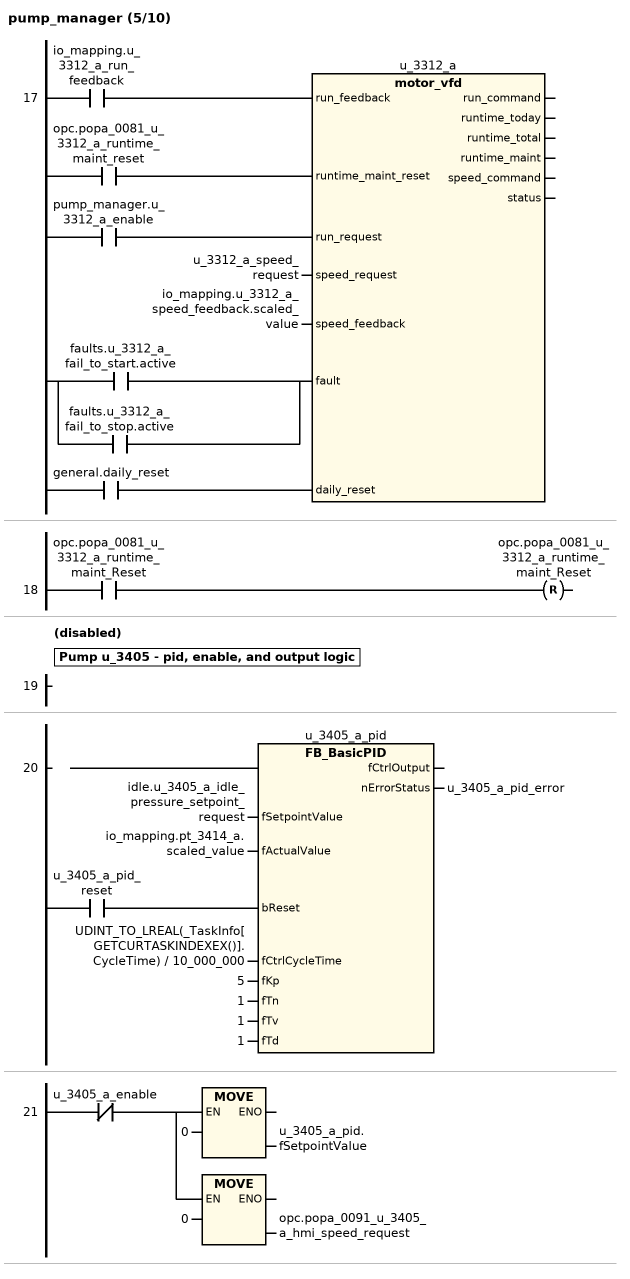
// NETWORK 17
u_3312_a(
    run_feedback := io_mapping.u_3312_a_run_feedback,
    runtime_maint_reset := opc.popa_0081_u_3312_a_runtime_maint_reset,
    run_request := pump_manager.u_3312_a_enable,
    speed_request := u_3312_a_speed_request,
    speed_feedback := io_mapping.u_3312_a_speed_feedback.scaled_value,
    fault := faults.u_3312_a_fail_to_start.active OR faults.u_3312_a_fail_to_stop.active,
    daily_reset := general.daily_reset); // motor_vfd

// NETWORK 18
opc.popa_0081_u_3312_a_runtime_maint_Reset R= opc.popa_0081_u_3312_a_runtime_maint_Reset;

// NETWORK 19 (disabled)
// label: Pump u_3405 - pid, enable, and output logic

// NETWORK 20
u_3405_a_pid(
    fSetpointValue := idle.u_3405_a_idle_pressure_setpoint_request,
    fActualValue := io_mapping.pt_3414_a.scaled_value,
    bReset := u_3405_a_pid_reset,
    fCtrlCycleTime := UDINT_TO_LREAL(_TaskInfo[GETCURTASKINDEXEX()].CycleTime) / 10_000_000,
    fKp := 5,
    fTn := 1,
    fTv := 1,
    fTd := 1,
    nErrorStatus => u_3405_a_pid_error); // FB_BasicPID

// NETWORK 21
_w16 := NOT u_3405_a_enable;
IF _w16 THEN u_3405_a_pid.fSetpointValue := 0; END_IF
IF _w16 THEN opc.popa_0091_u_3405_a_hmi_speed_request := 0; END_IF

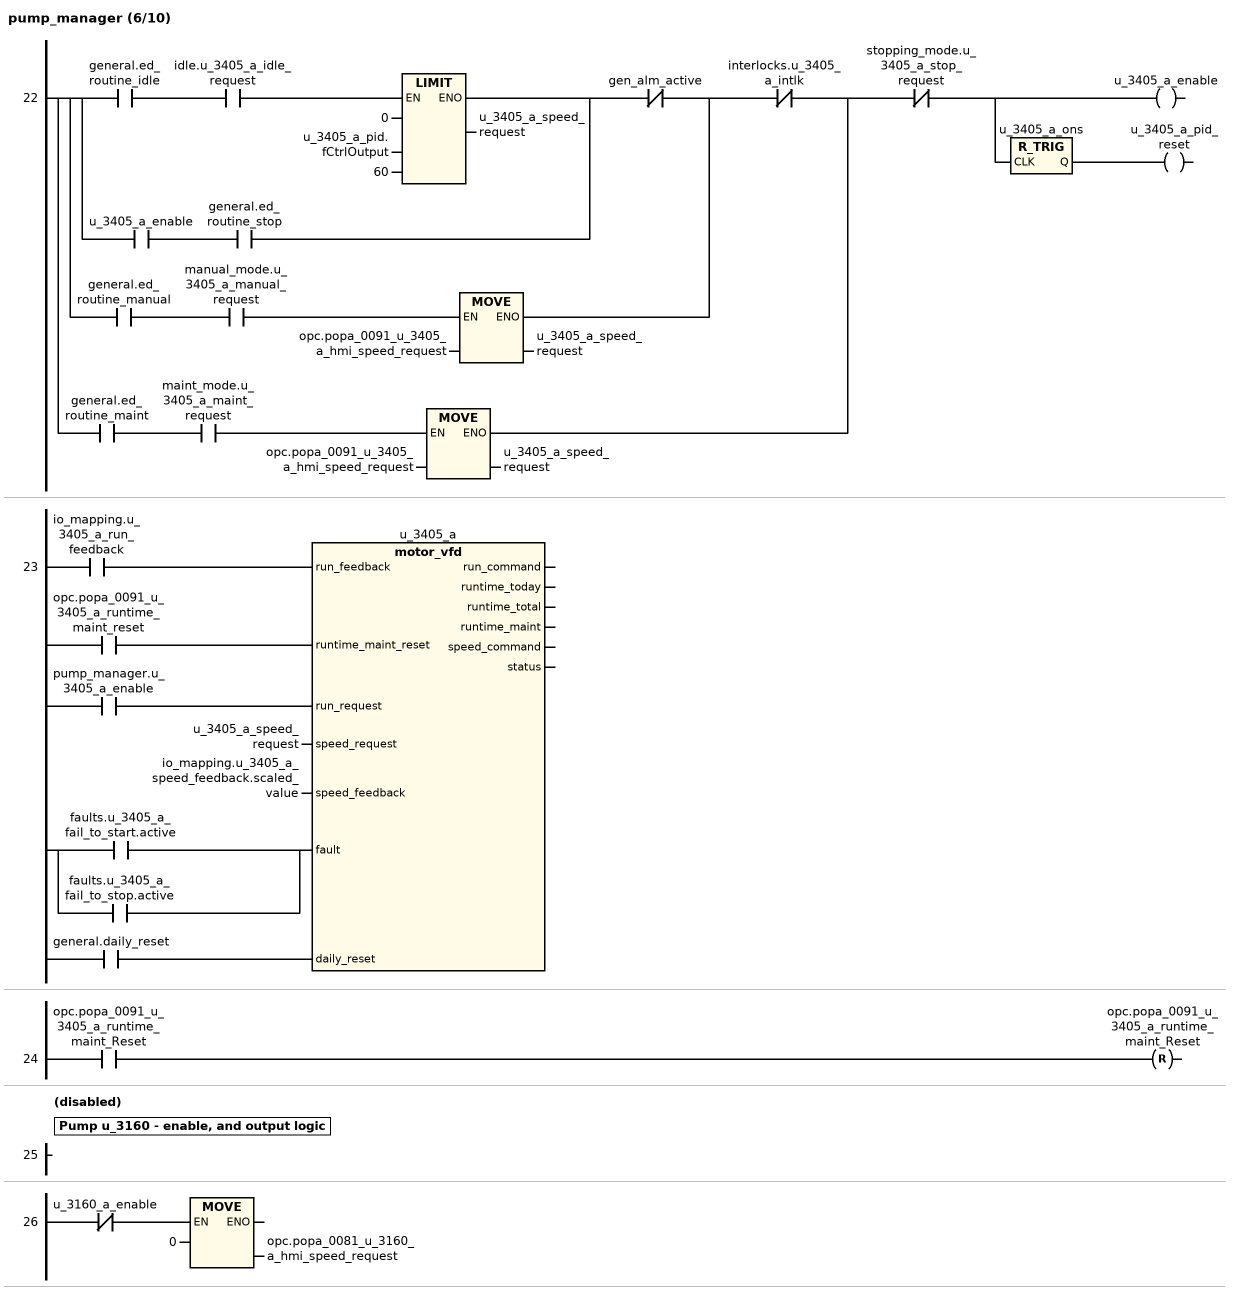
// NETWORK 22
_w17 := general.ed_routine_idle AND idle.u_3405_a_idle_request;
IF _w17 THEN u_3405_a_speed_request := LIMIT(0, u_3405_a_pid.fCtrlOutput, 60); END_IF
_w18 := general.ed_routine_manual AND manual_mode.u_3405_a_manual_request;
IF _w18 THEN u_3405_a_speed_request := opc.popa_0091_u_3405_a_hmi_speed_request; END_IF
_w19 := general.ed_routine_maint AND maint_mode.u_3405_a_maint_request;
IF _w19 THEN u_3405_a_speed_request := opc.popa_0091_u_3405_a_hmi_speed_request; END_IF
_w20 := (((_w17 OR u_3405_a_enable AND general.ed_routine_stop) AND NOT gen_alm_active OR _w18) AND NOT interlocks.u_3405_a_intlk OR _w19) AND NOT stopping_mode.u_3405_a_stop_request;
u_3405_a_enable := _w20;
u_3405_a_ons(CLK := _w20); // R_TRIG
u_3405_a_pid_reset := u_3405_a_ons.Q;

// NETWORK 23
u_3405_a(
    run_feedback := io_mapping.u_3405_a_run_feedback,
    runtime_maint_reset := opc.popa_0091_u_3405_a_runtime_maint_reset,
    run_request := pump_manager.u_3405_a_enable,
    speed_request := u_3405_a_speed_request,
    speed_feedback := io_mapping.u_3405_a_speed_feedback.scaled_value,
    fault := faults.u_3405_a_fail_to_start.active OR faults.u_3405_a_fail_to_stop.active,
    daily_reset := general.daily_reset); // motor_vfd

// NETWORK 24
opc.popa_0091_u_3405_a_runtime_maint_Reset R= opc.popa_0091_u_3405_a_runtime_maint_Reset;

// NETWORK 25 (disabled)
// label: Pump u_3160 - enable, and output logic

// NETWORK 26
IF NOT u_3160_a_enable THEN opc.popa_0081_u_3160_a_hmi_speed_request := 0; END_IF

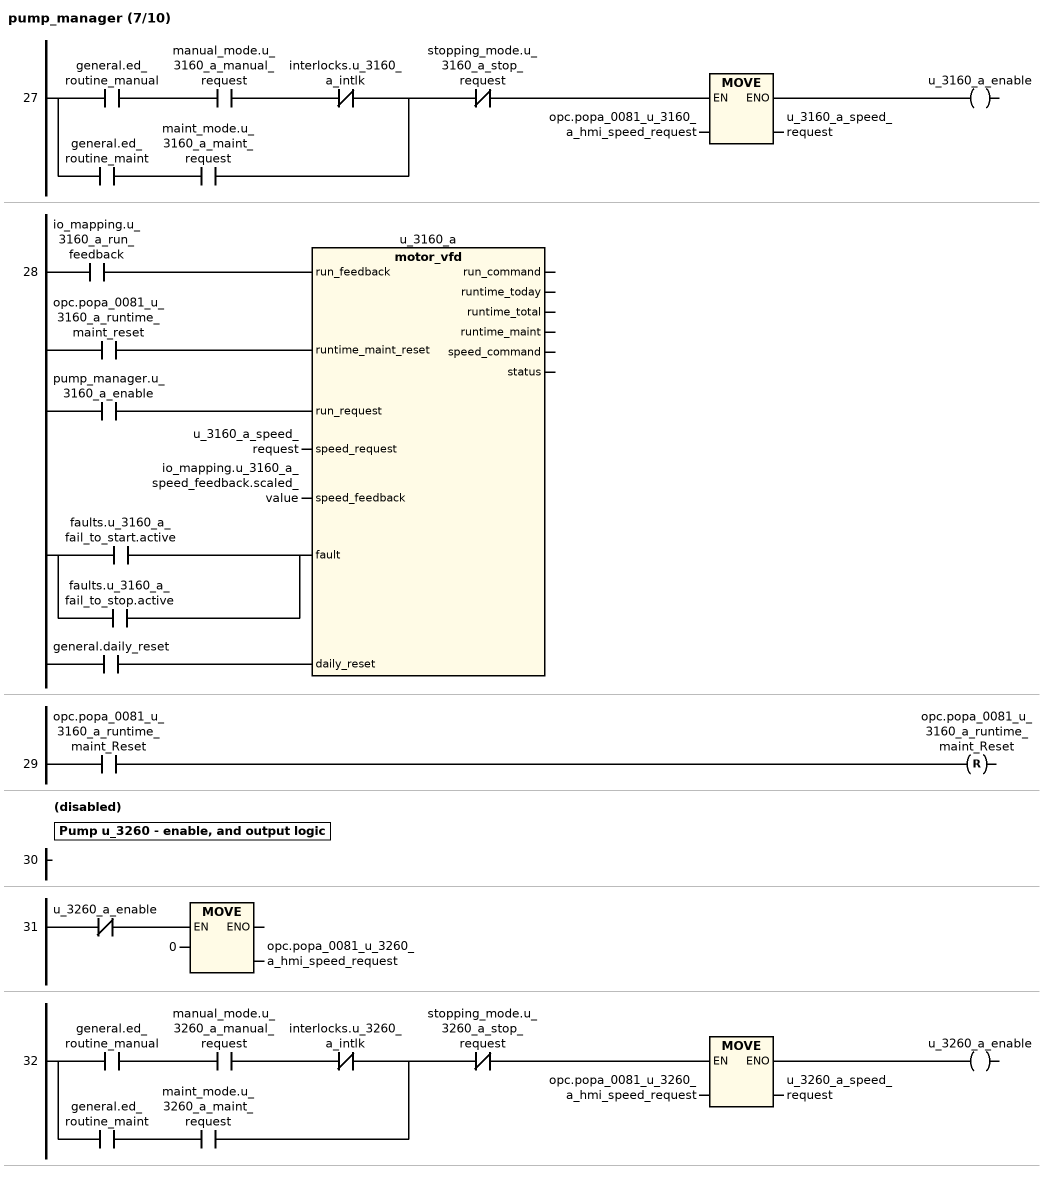
// NETWORK 27
_w21 := (general.ed_routine_manual AND manual_mode.u_3160_a_manual_request AND NOT interlocks.u_3160_a_intlk OR general.ed_routine_maint AND maint_mode.u_3160_a_maint_request) AND NOT stopping_mode.u_3160_a_stop_request;
IF _w21 THEN u_3160_a_speed_request := opc.popa_0081_u_3160_a_hmi_speed_request; END_IF
u_3160_a_enable := _w21;

// NETWORK 28
u_3160_a(
    run_feedback := io_mapping.u_3160_a_run_feedback,
    runtime_maint_reset := opc.popa_0081_u_3160_a_runtime_maint_reset,
    run_request := pump_manager.u_3160_a_enable,
    speed_request := u_3160_a_speed_request,
    speed_feedback := io_mapping.u_3160_a_speed_feedback.scaled_value,
    fault := faults.u_3160_a_fail_to_start.active OR faults.u_3160_a_fail_to_stop.active,
    daily_reset := general.daily_reset); // motor_vfd

// NETWORK 29
opc.popa_0081_u_3160_a_runtime_maint_Reset R= opc.popa_0081_u_3160_a_runtime_maint_Reset;

// NETWORK 30 (disabled)
// label: Pump u_3260 - enable, and output logic

// NETWORK 31
IF NOT u_3260_a_enable THEN opc.popa_0081_u_3260_a_hmi_speed_request := 0; END_IF

// NETWORK 32
_w22 := (general.ed_routine_manual AND manual_mode.u_3260_a_manual_request AND NOT interlocks.u_3260_a_intlk OR general.ed_routine_maint AND maint_mode.u_3260_a_maint_request) AND NOT stopping_mode.u_3260_a_stop_request;
IF _w22 THEN u_3260_a_speed_request := opc.popa_0081_u_3260_a_hmi_speed_request; END_IF
u_3260_a_enable := _w22;

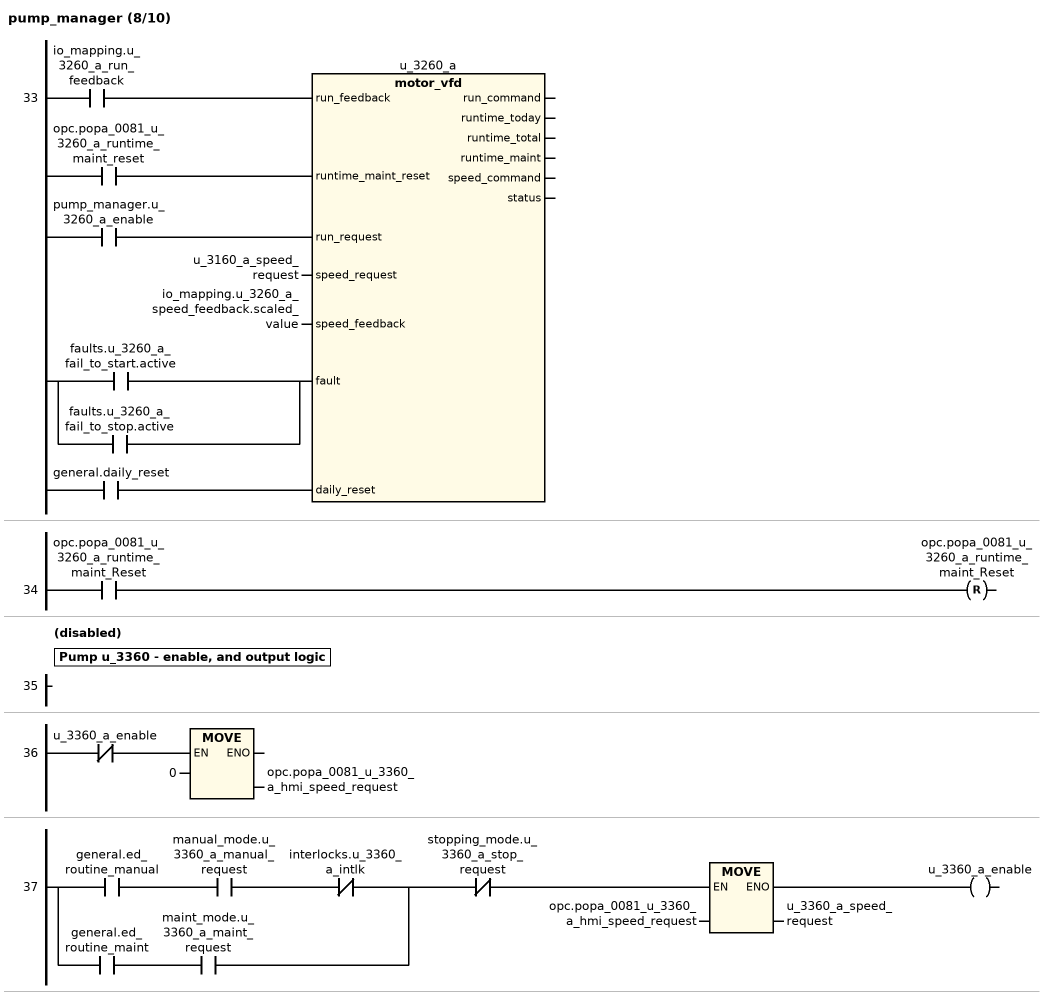
// NETWORK 33
u_3260_a(
    run_feedback := io_mapping.u_3260_a_run_feedback,
    runtime_maint_reset := opc.popa_0081_u_3260_a_runtime_maint_reset,
    run_request := pump_manager.u_3260_a_enable,
    speed_request := u_3160_a_speed_request,
    speed_feedback := io_mapping.u_3260_a_speed_feedback.scaled_value,
    fault := faults.u_3260_a_fail_to_start.active OR faults.u_3260_a_fail_to_stop.active,
    daily_reset := general.daily_reset); // motor_vfd

// NETWORK 34
opc.popa_0081_u_3260_a_runtime_maint_Reset R= opc.popa_0081_u_3260_a_runtime_maint_Reset;

// NETWORK 35 (disabled)
// label: Pump u_3360 - enable, and output logic

// NETWORK 36
IF NOT u_3360_a_enable THEN opc.popa_0081_u_3360_a_hmi_speed_request := 0; END_IF

// NETWORK 37
_w23 := (general.ed_routine_manual AND manual_mode.u_3360_a_manual_request AND NOT interlocks.u_3360_a_intlk OR general.ed_routine_maint AND maint_mode.u_3360_a_maint_request) AND NOT stopping_mode.u_3360_a_stop_request;
IF _w23 THEN u_3360_a_speed_request := opc.popa_0081_u_3360_a_hmi_speed_request; END_IF
u_3360_a_enable := _w23;

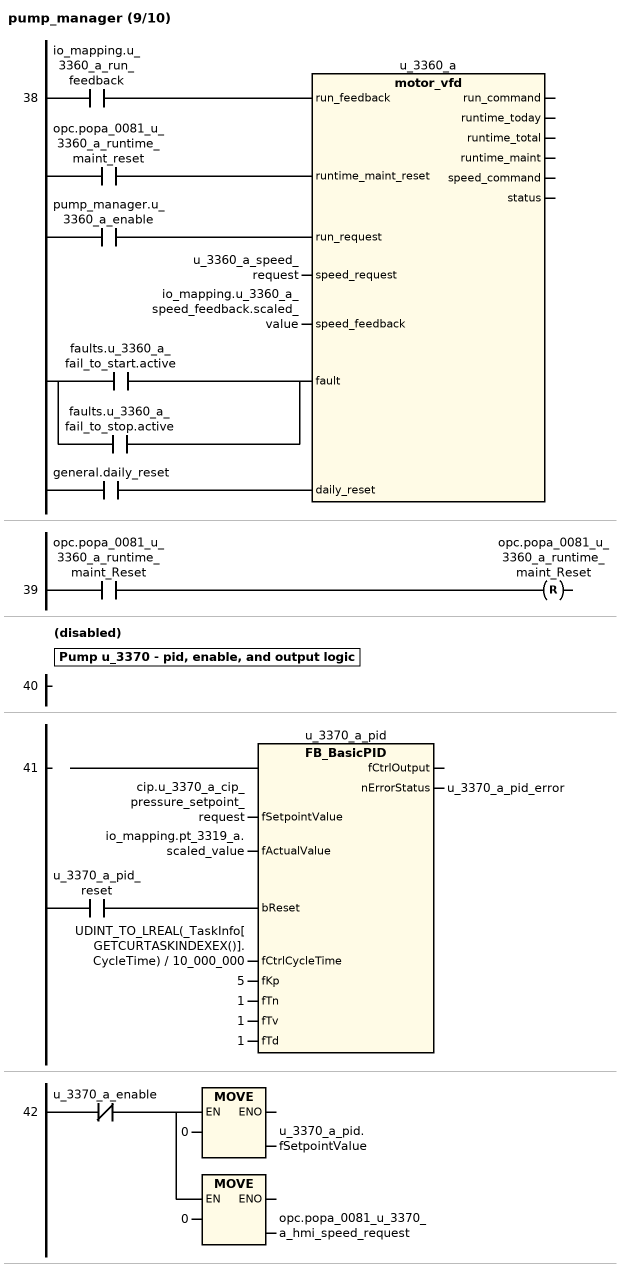
// NETWORK 38
u_3360_a(
    run_feedback := io_mapping.u_3360_a_run_feedback,
    runtime_maint_reset := opc.popa_0081_u_3360_a_runtime_maint_reset,
    run_request := pump_manager.u_3360_a_enable,
    speed_request := u_3360_a_speed_request,
    speed_feedback := io_mapping.u_3360_a_speed_feedback.scaled_value,
    fault := faults.u_3360_a_fail_to_start.active OR faults.u_3360_a_fail_to_stop.active,
    daily_reset := general.daily_reset); // motor_vfd

// NETWORK 39
opc.popa_0081_u_3360_a_runtime_maint_Reset R= opc.popa_0081_u_3360_a_runtime_maint_Reset;

// NETWORK 40 (disabled)
// label: Pump u_3370 - pid, enable, and output logic

// NETWORK 41
u_3370_a_pid(
    fSetpointValue := cip.u_3370_a_cip_pressure_setpoint_request,
    fActualValue := io_mapping.pt_3319_a.scaled_value,
    bReset := u_3370_a_pid_reset,
    fCtrlCycleTime := UDINT_TO_LREAL(_TaskInfo[GETCURTASKINDEXEX()].CycleTime) / 10_000_000,
    fKp := 5,
    fTn := 1,
    fTv := 1,
    fTd := 1,
    nErrorStatus => u_3370_a_pid_error); // FB_BasicPID

// NETWORK 42
_w24 := NOT u_3370_a_enable;
IF _w24 THEN u_3370_a_pid.fSetpointValue := 0; END_IF
IF _w24 THEN opc.popa_0081_u_3370_a_hmi_speed_request := 0; END_IF

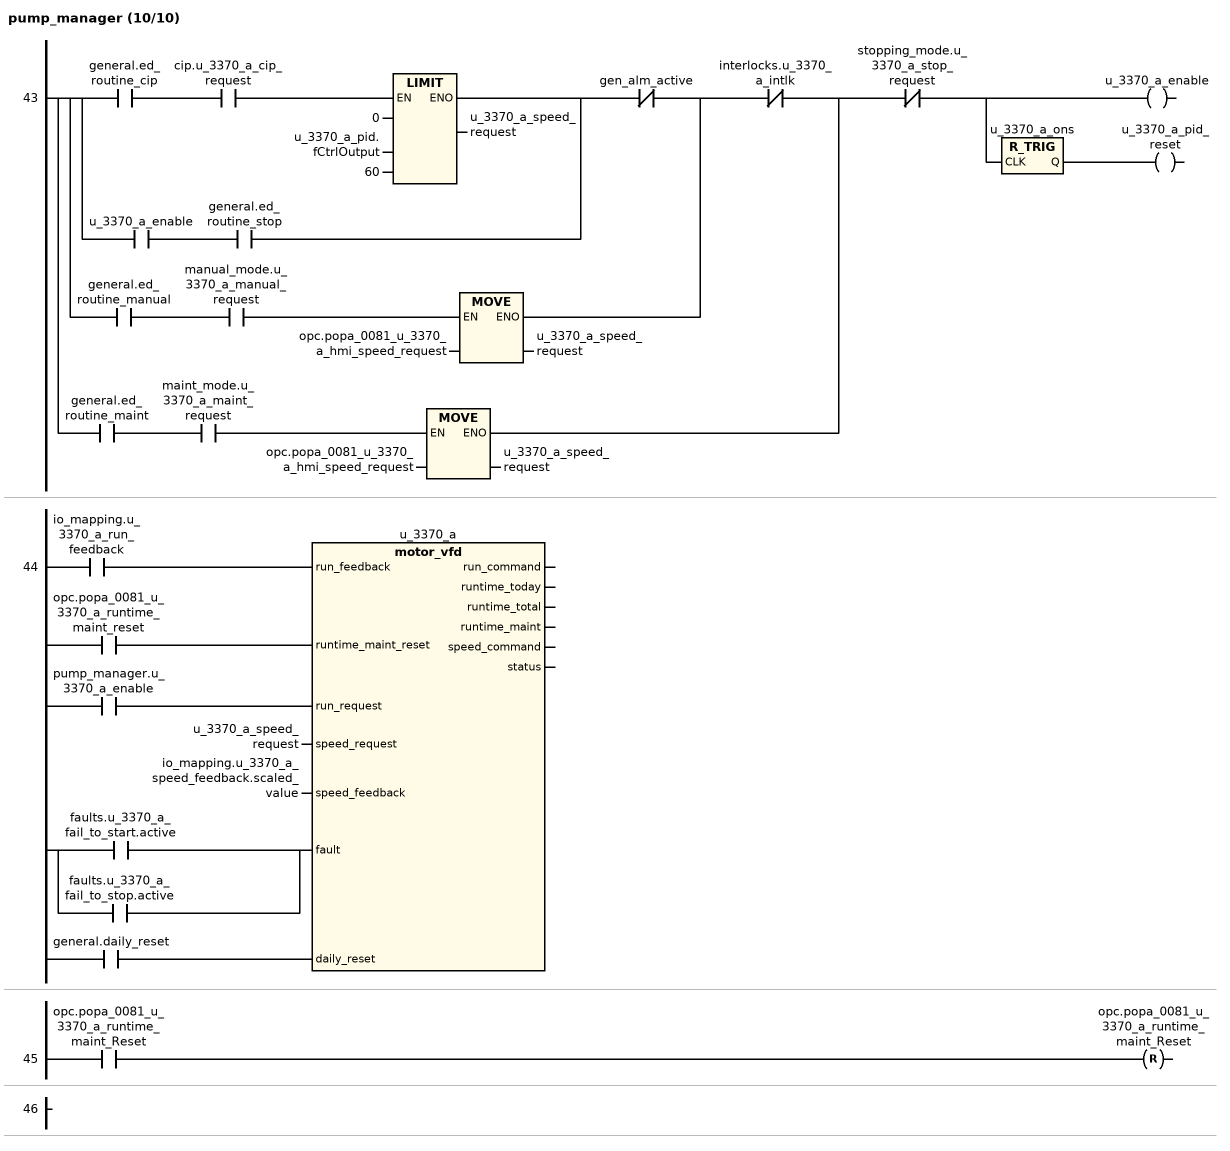
// NETWORK 43
_w25 := general.ed_routine_cip AND cip.u_3370_a_cip_request;
IF _w25 THEN u_3370_a_speed_request := LIMIT(0, u_3370_a_pid.fCtrlOutput, 60); END_IF
_w26 := general.ed_routine_manual AND manual_mode.u_3370_a_manual_request;
IF _w26 THEN u_3370_a_speed_request := opc.popa_0081_u_3370_a_hmi_speed_request; END_IF
_w27 := general.ed_routine_maint AND maint_mode.u_3370_a_maint_request;
IF _w27 THEN u_3370_a_speed_request := opc.popa_0081_u_3370_a_hmi_speed_request; END_IF
_w28 := (((_w25 OR u_3370_a_enable AND general.ed_routine_stop) AND NOT gen_alm_active OR _w26) AND NOT interlocks.u_3370_a_intlk OR _w27) AND NOT stopping_mode.u_3370_a_stop_request;
u_3370_a_enable := _w28;
u_3370_a_ons(CLK := _w28); // R_TRIG
u_3370_a_pid_reset := u_3370_a_ons.Q;

// NETWORK 44
u_3370_a(
    run_feedback := io_mapping.u_3370_a_run_feedback,
    runtime_maint_reset := opc.popa_0081_u_3370_a_runtime_maint_reset,
    run_request := pump_manager.u_3370_a_enable,
    speed_request := u_3370_a_speed_request,
    speed_feedback := io_mapping.u_3370_a_speed_feedback.scaled_value,
    fault := faults.u_3370_a_fail_to_start.active OR faults.u_3370_a_fail_to_stop.active,
    daily_reset := general.daily_reset); // motor_vfd

// NETWORK 45
opc.popa_0081_u_3370_a_runtime_maint_Reset R= opc.popa_0081_u_3370_a_runtime_maint_Reset;

// NETWORK 46

END_PROGRAM

// ---- POUs/idle.TcPOU
PROGRAM idle
VAR
	ed_routine_idle: BOOL;
	redox_doser_idle_enable: BOOL;
	
	tmr_idle_pumps: TON;
	u_3112_idle_request: BOOL;
	u_3312_idle_request: BOOL;
	u_3405_idle_request: BOOL;
	u_3212_idle_request: BOOL;
	tmr_idle_pump_delay: TON;
	u_3112_running: BOOL;
	u_3112_speed_ref: INT;
	u_3112_sp: REAL;
	salt_pressure_actual: REAL;
	u_3112_ready: BOOL;
	u_3212_running: BOOL;
	u_3212_ready: BOOL;
	u_3312_ready: BOOL;
	u_3312_running: BOOL;
	u_3405_running: BOOL;
	u_3405_ready: BOOL;
	stack_power_enable: BOOL;
	nv_3110_open_request: BOOL;
	nv_3210_open_request: BOOL;
	nv_3310_open_request: BOOL;
	nv_3110_open_feedback: BOOL;
	nv_3210_open_feedback: BOOL;
	nv_3310_open_feedback: BOOL;
	nv_3110_idle_request: BOOL;
	nv_3210_idle_request: BOOL;
	nv_3310_idle_request: BOOL;
	nv_3135_idle_request: BOOL;
	nv_3235_idle_request: BOOL;
	nv_3335_idle_request: BOOL;
	nv_3372_idle_request: BOOL;
	nv_3162_idle_request: BOOL;

	idle_stack_power_enable: BOOL;
	idle_TEMP_BIT: BOOL;
	tmr_idle_valye_delay: TON;
	tmr_idle_valve_delay: TON;
	tmr_idle_valve_delay_et: TIME;
	tmr_idle_valve_delay_pt: TIME := T#20S;
	tmr_idle_valve_delay_q: BOOL;
	u_3112_idle_pressure_setpoint_request: REAL;
	u_3212_idle_pressure_setpoint_request: REAL;
	u_3312_idle_pressure_setpoint_request: REAL;
	u_3405_idle_pressure_setpoint_request: REAL;
	idle_stable: BOOL;
	av_3148_idle_position_request: REAL;
	av_3248_idle_position_request: REAL;
	av_3348_idle_position_request: REAL;
	redox_pressure_calculation: REAL;
	redox_idle_pressure_sp_request: REAL;
	idle_startup_ons: R_TRIG;
END_VAR
VAR // added by the converter: edge detectors and wires of the graphical bodies
    _w1, _w2, _w3, _w4 : BOOL;
END_VAR

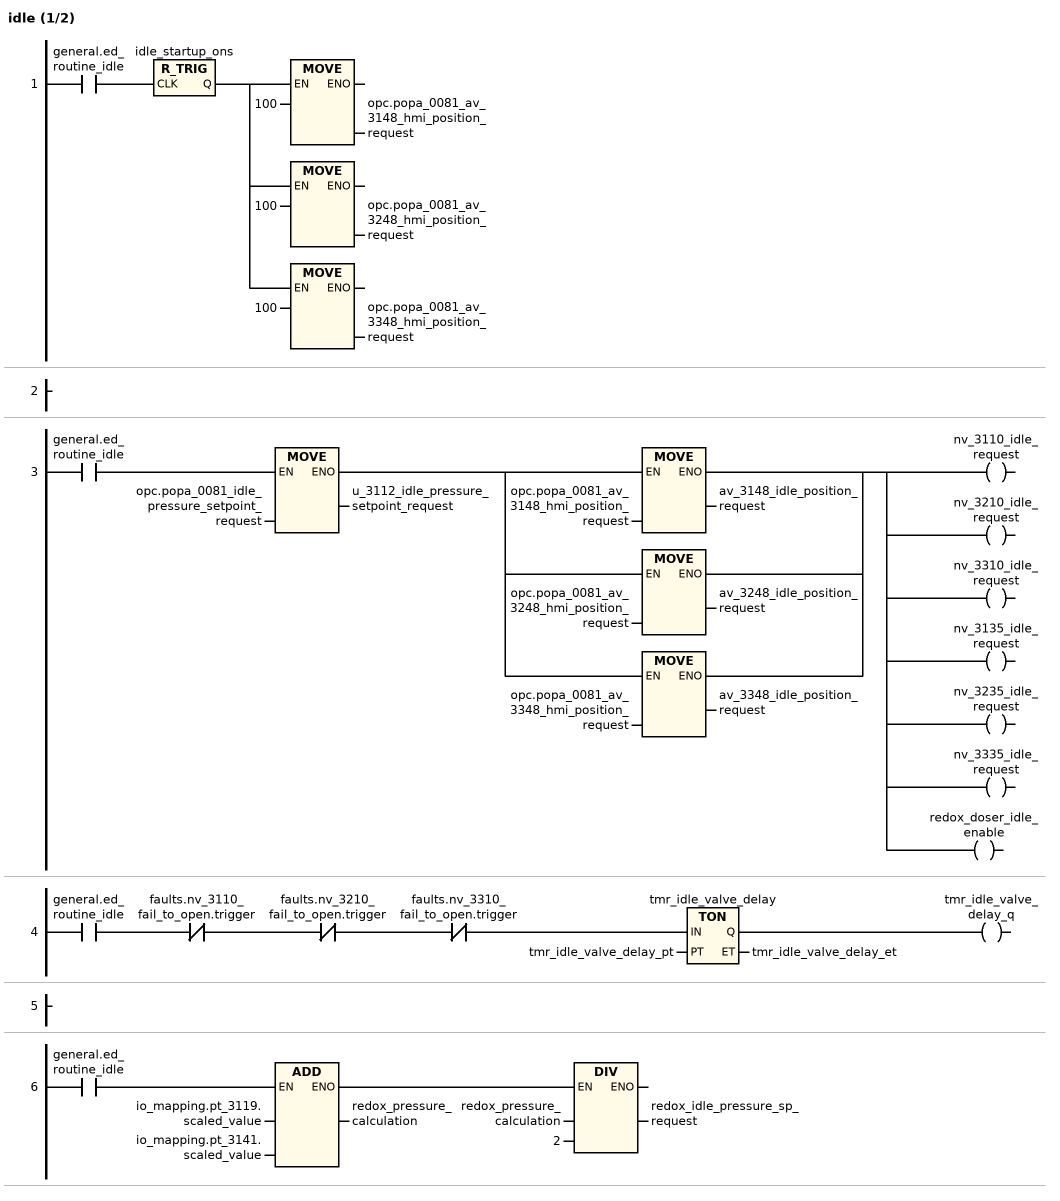
// NETWORK 1
idle_startup_ons(CLK := general.ed_routine_idle); // R_TRIG
IF idle_startup_ons.Q THEN opc.popa_0081_av_3148_hmi_position_request := 100; END_IF
IF idle_startup_ons.Q THEN opc.popa_0081_av_3248_hmi_position_request := 100; END_IF
IF idle_startup_ons.Q THEN opc.popa_0081_av_3348_hmi_position_request := 100; END_IF

// NETWORK 2

// NETWORK 3
_w1 := general.ed_routine_idle;
IF _w1 THEN u_3112_idle_pressure_setpoint_request := opc.popa_0081_idle_pressure_setpoint_request; END_IF
IF _w1 THEN av_3148_idle_position_request := opc.popa_0081_av_3148_hmi_position_request; END_IF
IF _w1 THEN av_3248_idle_position_request := opc.popa_0081_av_3248_hmi_position_request; END_IF
IF _w1 THEN av_3348_idle_position_request := opc.popa_0081_av_3348_hmi_position_request; END_IF
_w2 := _w1 OR (_w1 OR _w1);
nv_3110_idle_request := _w2;
nv_3210_idle_request := _w2;
nv_3310_idle_request := _w2;
nv_3135_idle_request := _w2;
nv_3235_idle_request := _w2;
nv_3335_idle_request := _w2;
redox_doser_idle_enable := _w2;

// NETWORK 4
tmr_idle_valve_delay(
    IN := general.ed_routine_idle AND NOT faults.nv_3110_fail_to_open.trigger AND NOT faults.nv_3210_fail_to_open.trigger AND NOT faults.nv_3310_fail_to_open.trigger,
    PT := tmr_idle_valve_delay_pt,
    ET => tmr_idle_valve_delay_et); // TON
tmr_idle_valve_delay_q := tmr_idle_valve_delay.Q;

// NETWORK 5

// NETWORK 6
_w3 := general.ed_routine_idle;
IF _w3 THEN redox_pressure_calculation := io_mapping.pt_3119.scaled_value + io_mapping.pt_3141.scaled_value; END_IF
IF _w3 THEN redox_idle_pressure_sp_request := redox_pressure_calculation / 2; END_IF

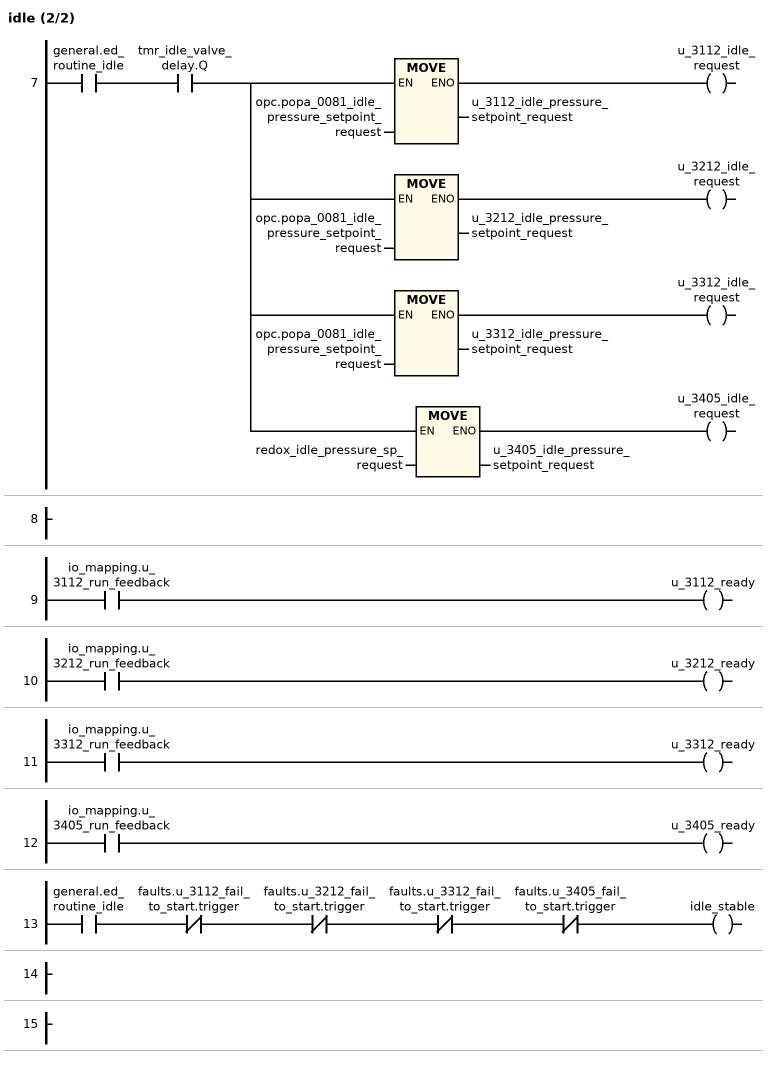
// NETWORK 7
_w4 := general.ed_routine_idle AND tmr_idle_valve_delay.Q;
IF _w4 THEN u_3112_idle_pressure_setpoint_request := opc.popa_0081_idle_pressure_setpoint_request; END_IF
u_3112_idle_request := _w4;
IF _w4 THEN u_3212_idle_pressure_setpoint_request := opc.popa_0081_idle_pressure_setpoint_request; END_IF
u_3212_idle_request := _w4;
IF _w4 THEN u_3312_idle_pressure_setpoint_request := opc.popa_0081_idle_pressure_setpoint_request; END_IF
u_3312_idle_request := _w4;
IF _w4 THEN u_3405_idle_pressure_setpoint_request := redox_idle_pressure_sp_request; END_IF
u_3405_idle_request := _w4;

// NETWORK 8

// NETWORK 9
u_3112_ready := io_mapping.u_3112_run_feedback;

// NETWORK 10
u_3212_ready := io_mapping.u_3212_run_feedback;

// NETWORK 11
u_3312_ready := io_mapping.u_3312_run_feedback;

// NETWORK 12
u_3405_ready := io_mapping.u_3405_run_feedback;

// NETWORK 13
idle_stable := general.ed_routine_idle AND NOT faults.u_3112_fail_to_start.trigger AND NOT faults.u_3212_fail_to_start.trigger AND NOT faults.u_3312_fail_to_start.trigger AND NOT faults.u_3405_fail_to_start.trigger;

// NETWORK 14

// NETWORK 15

END_PROGRAM

// ---- POUs/io_mapping.TcPOU
PROGRAM io_mapping
VAR PERSISTENT
//---Field Instrumentation-----------------------------------------------------------------------------------------------
    //Analog input function block
	cpt_3144_a: analog_scaling;
	
	cct_3120_a : analog_scaling;
	cct_3220_a : analog_scaling;
	cct_3320_a : analog_scaling;
	cct_3142_a : analog_scaling;
	cct_3242_a : analog_scaling;
	cct_3342_a : analog_scaling;
	
	ft_3122_a : analog_scaling;
	ft_3222_a : analog_scaling;
	ft_3322_a : analog_scaling;
	
	lt_3102_a : analog_scaling;
	lt_3202_a : analog_scaling;
	lt_3302_a : analog_scaling;
	lt_3153_a : analog_scaling;
	lt_3253_a : analog_scaling;
	lt_3353_a : analog_scaling;
	lt_3402_a : analog_scaling;
	
    pt_3119_a : analog_scaling;
	pt_3219_a : analog_scaling;
	pt_3319_a : analog_scaling;
	pt_3141_a : analog_scaling;
	pt_3241_a : analog_scaling;
	pt_3341_a : analog_scaling;
	pt_3428_a : analog_scaling;
	pt_3414_a : analog_scaling;
	
	tt_3118_a : analog_scaling;
	tt_3218_a : analog_scaling;
	tt_3318_a : analog_scaling;
	tt_3140_a : analog_scaling;
	tt_3240_a : analog_scaling;
	tt_3340_a : analog_scaling;
	tt_3432_a : analog_scaling;

	//Motor vfd speed feedback
	u_3112_a_speed_feedback : analog_scaling;
	u_3212_a_speed_feedback : analog_scaling;
	u_3312_a_speed_feedback : analog_scaling;
	u_3160_a_speed_feedback : analog_scaling;
	u_3260_a_speed_feedback : analog_scaling;
	u_3360_a_speed_feedback : analog_scaling;
	u_3370_a_speed_feedback : analog_scaling;
	u_3405_a_speed_feedback : analog_scaling;	
	
	//Analog valve position feedback
	av_3148_a_position_feedback : analog_scaling;
	av_3248_a_position_feedback : analog_scaling;
	av_3348_a_position_feedback : analog_scaling;
    //Analog input raw input, mapped to a physical input
    cpt_3144_a_raw_input AT %I* : INT;
	{attribute 'TcLinkTo' := 'TIID^Device 1 (EtherCAT)^Term 20 (EK1100-0018)^Term 24 (EL3058)^AI Standard Channel 1^Value'}
	cct_3120_a_raw_input AT %I* : INT;
	{attribute 'TcLinkTo' := 'TIID^Device 1 (EtherCAT)^Term 20 (EK1100-0018)^Term 24 (EL3058)^AI Standard Channel 2^Value'}
	cct_3220_a_raw_input AT %I* : INT;
	{attribute 'TcLinkTo' := 'TIID^Device 1 (EtherCAT)^Term 20 (EK1100-0018)^Term 24 (EL3058)^AI Standard Channel 3^Value'}
	cct_3320_a_raw_input AT %I* : INT;
	{attribute 'TcLinkTo' := 'TIID^Device 1 (EtherCAT)^Term 20 (EK1100-0018)^Term 24 (EL3058)^AI Standard Channel 4^Value'}
	cct_3142_a_raw_input AT %I* : INT;
	{attribute 'TcLinkTo' := 'TIID^Device 1 (EtherCAT)^Term 20 (EK1100-0018)^Term 24 (EL3058)^AI Standard Channel 5^Value'}
	cct_3242_a_raw_input AT %I* : INT;
	{attribute 'TcLinkTo' := 'TIID^Device 1 (EtherCAT)^Term 20 (EK1100-0018)^Term 24 (EL3058)^AI Standard Channel 6^Value'}
	cct_3342_a_raw_input AT %I* : INT;
	
	{attribute 'TcLinkTo' := 'TIID^Device 1 (EtherCAT)^Term 20 (EK1100-0018)^Term 25 (EL3058)^AI Standard Channel 1^Value'}
	ft_3122_a_raw_input AT %I* : INT;
	{attribute 'TcLinkTo' := 'TIID^Device 1 (EtherCAT)^Term 20 (EK1100-0018)^Term 25 (EL3058)^AI Standard Channel 2^Value'}
	ft_3222_a_raw_input AT %I* : INT;
	{attribute 'TcLinkTo' := 'TIID^Device 1 (EtherCAT)^Term 20 (EK1100-0018)^Term 25 (EL3058)^AI Standard Channel 3^Value'}
	ft_3322_a_raw_input AT %I* : INT;
	
	{attribute 'TcLinkTo' := 'TIID^Device 1 (EtherCAT)^Term 20 (EK1100-0018)^Term 21 (EL3058)^AI Standard Channel 1^Value'}
	pt_3119_a_raw_input AT %I* : INT;
	{attribute 'TcLinkTo' := 'TIID^Device 1 (EtherCAT)^Term 20 (EK1100-0018)^Term 21 (EL3058)^AI Standard Channel 2^Value'}
	pt_3219_a_raw_input AT %I* : INT;
	{attribute 'TcLinkTo' := 'TIID^Device 1 (EtherCAT)^Term 20 (EK1100-0018)^Term 21 (EL3058)^AI Standard Channel 3^Value'}
	pt_3319_a_raw_input AT %I* : INT;
	{attribute 'TcLinkTo' := 'TIID^Device 1 (EtherCAT)^Term 20 (EK1100-0018)^Term 21 (EL3058)^AI Standard Channel 4^Value'}
	pt_3141_a_raw_input AT %I* : INT;
	{attribute 'TcLinkTo' := 'TIID^Device 1 (EtherCAT)^Term 20 (EK1100-0018)^Term 21 (EL3058)^AI Standard Channel 5^Value'}
	pt_3241_a_raw_input AT %I* : INT;
	{attribute 'TcLinkTo' := 'TIID^Device 1 (EtherCAT)^Term 20 (EK1100-0018)^Term 21 (EL3058)^AI Standard Channel 6^Value'}
	pt_3341_a_raw_input AT %I* : INT;
	{attribute 'TcLinkTo' := 'TIID^Device 1 (EtherCAT)^Term 40 (EK1100)^Term 41 (EL3058)^AI Standard Channel 4^Value'}
	pt_3428_a_raw_input AT %I* : INT;
	{attribute 'TcLinkTo' := 'TIID^Device 1 (EtherCAT)^Term 40 (EK1100)^Term 41 (EL3058)^AI Standard Channel 5^Value'}
	pt_3414_a_raw_input AT %I* : INT;
	
	{attribute 'TcLinkTo' := 'TIID^Device 1 (EtherCAT)^Term 20 (EK1100-0018)^Term 23 (EL3058)^AI Standard Channel 3^Value'}
	lt_3102_a_raw_input AT %I* : INT;
	{attribute 'TcLinkTo' := 'TIID^Device 1 (EtherCAT)^Term 20 (EK1100-0018)^Term 23 (EL3058)^AI Standard Channel 4^Value'}
	lt_3202_a_raw_input AT %I* : INT;
	{attribute 'TcLinkTo' := 'TIID^Device 1 (EtherCAT)^Term 20 (EK1100-0018)^Term 23 (EL3058)^AI Standard Channel 5^Value'}
	lt_3302_a_raw_input AT %I* : INT;
	{attribute 'TcLinkTo' := 'TIID^Device 1 (EtherCAT)^Term 20 (EK1100-0018)^Term 23 (EL3058)^AI Standard Channel 6^Value'}
	lt_3153_a_raw_input AT %I* : INT;
	{attribute 'TcLinkTo' := 'TIID^Device 1 (EtherCAT)^Term 20 (EK1100-0018)^Term 23 (EL3058)^AI Standard Channel 7^Value'}
	lt_3253_a_raw_input AT %I* : INT;
	{attribute 'TcLinkTo' := 'TIID^Device 1 (EtherCAT)^Term 20 (EK1100-0018)^Term 23 (EL3058)^AI Standard Channel 8^Value'}
	lt_3353_a_raw_input AT %I* : INT;
	{attribute 'TcLinkTo' := 'TIID^Device 1 (EtherCAT)^Term 40 (EK1100)^Term 41 (EL3058)^AI Standard Channel 3^Value'}
	lt_3402_a_raw_input AT %I* : INT;
	
	{attribute 'TcLinkTo' := 'TIID^Device 1 (EtherCAT)^Term 20 (EK1100-0018)^Term 21 (EL3058)^AI Standard Channel 7^Value'}
	tt_3118_a_raw_input AT %I* : INT;
	{attribute 'TcLinkTo' := 'TIID^Device 1 (EtherCAT)^Term 20 (EK1100-0018)^Term 21 (EL3058)^AI Standard Channel 8^Value'}
	tt_3218_a_raw_input AT %I* : INT;
	{attribute 'TcLinkTo' := 'TIID^Device 1 (EtherCAT)^Term 20 (EK1100-0018)^Term 22 (EL3058)^AI Standard Channel 1^Value'}
	tt_3318_a_raw_input AT %I* : INT;
	{attribute 'TcLinkTo' := 'TIID^Device 1 (EtherCAT)^Term 20 (EK1100-0018)^Term 22 (EL3058)^AI Standard Channel 2^Value'}
	tt_3140_a_raw_input AT %I* : INT;
	{attribute 'TcLinkTo' := 'TIID^Device 1 (EtherCAT)^Term 20 (EK1100-0018)^Term 22 (EL3058)^AI Standard Channel 3^Value'}
	tt_3240_a_raw_input AT %I* : INT;
	{attribute 'TcLinkTo' := 'TIID^Device 1 (EtherCAT)^Term 20 (EK1100-0018)^Term 22 (EL3058)^AI Standard Channel 4^Value'}
	tt_3340_a_raw_input AT %I* : INT;
	{attribute 'TcLinkTo' := 'TIID^Device 1 (EtherCAT)^Term 40 (EK1100)^Term 41 (EL3058)^AI Standard Channel 2^Value'}
	tt_3432_a_raw_input AT %I* : INT;
	
//---Field Equipment:Pumps----------------------------------------------------------------------------------------------------------
	
	//Motor vfd run feedback, mapped to a physical input
	{attribute 'TcLinkTo' := 'TIID^Device 1 (EtherCAT)^Term 1 (EK1200)^Term 7 (EL1859)^Channel 2^Input'}
	u_3112_a_run_feedback AT %I* : BOOL;
	{attribute 'TcLinkTo' := 'TIID^Device 1 (EtherCAT)^Term 1 (EK1200)^Term 7 (EL1859)^Channel 4^Input'}
	u_3212_a_run_feedback AT %I* : BOOL;
	{attribute 'TcLinkTo' := 'TIID^Device 1 (EtherCAT)^Term 1 (EK1200)^Term 7 (EL1859)^Channel 6^Input'}
	u_3312_a_run_feedback AT %I* : BOOL;
	{attribute 'TcLinkTo' := 'TIID^Device 1 (EtherCAT)^Term 1 (EK1200)^Term 7 (EL1859)^Channel 8^Input'}
	u_3160_a_run_feedback AT %I* : BOOL;
	{attribute 'TcLinkTo' := 'TIID^Device 1 (EtherCAT)^Term 1 (EK1200)^Term 8 (EL1859)^Channel 2^Input'}
	u_3260_a_run_feedback AT %I* : BOOL;
	{attribute 'TcLinkTo' := 'TIID^Device 1 (EtherCAT)^Term 1 (EK1200)^Term 8 (EL1859)^Channel 4^Input'}
	u_3360_a_run_feedback AT %I* : BOOL;
	{attribute 'TcLinkTo' := 'TIID^Device 1 (EtherCAT)^Term 1 (EK1200)^Term 8 (EL1859)^Channel 6^Input'}
	u_3370_a_run_feedback AT %I* : BOOL;
	{attribute 'TcLinkTo' := 'TIID^Device 1 (EtherCAT)^Term 40 (EK1100)^Term 43 (EL1859)^Channel 2^Input'}
	u_3405_a_run_feedback AT %I* : BOOL;
	
	//Motor Fault feedback
	{attribute 'TcLinkTo' := 'TIID^Device 1 (EtherCAT)^Term 1 (EK1200)^Term 7 (EL1859)^Channel 1^Input'}
	u_3112_a_fault_feedback AT %I* : BOOL;
	{attribute 'TcLinkTo' := 'TIID^Device 1 (EtherCAT)^Term 1 (EK1200)^Term 7 (EL1859)^Channel 3^Input'}
	u_3212_a_fault_feedback AT %I* : BOOL;
	{attribute 'TcLinkTo' := 'TIID^Device 1 (EtherCAT)^Term 1 (EK1200)^Term 7 (EL1859)^Channel 5^Input'}
	u_3312_a_fault_feedback AT %I* : BOOL;
	{attribute 'TcLinkTo' := 'TIID^Device 1 (EtherCAT)^Term 1 (EK1200)^Term 7 (EL1859)^Channel 7^Input'}
	u_3160_a_fault_feedback AT %I* : BOOL;
	{attribute 'TcLinkTo' := 'TIID^Device 1 (EtherCAT)^Term 1 (EK1200)^Term 8 (EL1859)^Channel 1^Input'}
	u_3260_a_fault_feedback AT %I* : BOOL;
	{attribute 'TcLinkTo' := 'TIID^Device 1 (EtherCAT)^Term 1 (EK1200)^Term 8 (EL1859)^Channel 3^Input'}
	u_3360_a_fault_feedback AT %I* : BOOL;
	{attribute 'TcLinkTo' := 'TIID^Device 1 (EtherCAT)^Term 1 (EK1200)^Term 8 (EL1859)^Channel 5^Input'}
	u_3370_a_fault_feedback AT %I* : BOOL;
	{attribute 'TcLinkTo' := 'TIID^Device 1 (EtherCAT)^Term 40 (EK1100)^Term 43 (EL1859)^Channel 1^Input'}
	u_3405_a_fault_feedback AT %I* : BOOL;
	
	
	
	

	
	//Motor vfd speed feedback raw input
	{attribute 'TcLinkTo' := 'TIID^Device 1 (EtherCAT)^Term 1 (EK1200)^Term 2 (EL3058)^AI Standard Channel 1^Value'}
	u_3112_a_speed_feedback_raw_input AT %I* : INT;
	{attribute 'TcLinkTo' := 'TIID^Device 1 (EtherCAT)^Term 1 (EK1200)^Term 2 (EL3058)^AI Standard Channel 2^Value'}
	u_3212_a_speed_feedback_raw_input AT %I* : INT;
	{attribute 'TcLinkTo' := 'TIID^Device 1 (EtherCAT)^Term 1 (EK1200)^Term 2 (EL3058)^AI Standard Channel 3^Value'}
	u_3312_a_speed_feedback_raw_input AT %I* : INT;
	{attribute 'TcLinkTo' := 'TIID^Device 1 (EtherCAT)^Term 1 (EK1200)^Term 2 (EL3058)^AI Standard Channel 4^Value'}
	u_3160_a_speed_feedback_raw_input AT %I* : INT;
	{attribute 'TcLinkTo' := 'TIID^Device 1 (EtherCAT)^Term 1 (EK1200)^Term 2 (EL3058)^AI Standard Channel 5^Value'}
	u_3260_a_speed_feedback_raw_input AT %I* : INT;
	{attribute 'TcLinkTo' := 'TIID^Device 1 (EtherCAT)^Term 1 (EK1200)^Term 2 (EL3058)^AI Standard Channel 6^Value'}
	u_3360_a_speed_feedback_raw_input AT %I* : INT;
	{attribute 'TcLinkTo' := 'TIID^Device 1 (EtherCAT)^Term 1 (EK1200)^Term 2 (EL3058)^AI Standard Channel 7^Value'}
	u_3370_a_speed_feedback_raw_input AT %I* : INT;
	{attribute 'TcLinkTo' := 'TIID^Device 1 (EtherCAT)^Term 40 (EK1100)^Term 41 (EL3058)^AI Standard Channel 1^Value'}
	u_3405_a_speed_feedback_raw_input AT %I* : INT;
	
//--Field Equipent: Valves---------------------------------------------------------------------------------------------------------------
	

	//Analog valve position feedback raw input
	{attribute 'TcLinkTo' := 'TIID^Device 1 (EtherCAT)^Term 20 (EK1100-0018)^Term 22 (EL3058)^AI Standard Channel 8^Value'}
	av_3148_a_position_feedback_raw_input AT %I* : INT;
	{attribute 'TcLinkTo' := 'TIID^Device 1 (EtherCAT)^Term 20 (EK1100-0018)^Term 23 (EL3058)^AI Standard Channel 1^Value'}
	av_3248_a_position_feedback_raw_input AT %I* : INT;
	{attribute 'TcLinkTo' := 'TIID^Device 1 (EtherCAT)^Term 20 (EK1100-0018)^Term 23 (EL3058)^AI Standard Channel 2^Value'}
	av_3348_a_position_feedback_raw_input AT %I* : INT;
	

	
	//Digital valve open feedback
	//{attribute 'TcLinkTo' := 'TIID^Device 1 (EtherCAT)^Term 31 (EK1914)^Term 32 (EL1859)^Channel 11^Output'}
	nv_3110_a_open_feedback AT %I* : BOOL;
	//{attribute 'TcLinkTo' := 'TIID^Device 1 (EtherCAT)^Term 31 (EK1914)^Term 32 (EL1859)^Channel 11^Output'}
	nv_3210_a_open_feedback AT %I* : BOOL;
	//{attribute 'TcLinkTo' := 'TIID^Device 1 (EtherCAT)^Term 31 (EK1914)^Term 32 (EL1859)^Channel 11^Output'}
	nv_3310_a_open_feedback AT %I* : BOOL;
	{attribute 'TcLinkTo' := 'TIID^Device 1 (EtherCAT)^Term 20 (EK1100-0018)^Term 28 (EL1859)^Channel 1^Input'}
	nv_3135_a_open_feedback AT %I* : BOOL;
	{attribute 'TcLinkTo' := 'TIID^Device 1 (EtherCAT)^Term 20 (EK1100-0018)^Term 28 (EL1859)^Channel 2^Input'}
	nv_3235_a_open_feedback AT %I* : BOOL;
	{attribute 'TcLinkTo' := 'TIID^Device 1 (EtherCAT)^Term 20 (EK1100-0018)^Term 28 (EL1859)^Channel 3^Input'}
	nv_3335_a_open_feedback AT %I* : BOOL;
	{attribute 'TcLinkTo' := 'TIID^Device 1 (EtherCAT)^Term 20 (EK1100-0018)^Term 28 (EL1859)^Channel 4^Input'}
	nv_3372_a_open_feedback AT %I* : BOOL;
	{attribute 'TcLinkTo' := 'TIID^Device 1 (EtherCAT)^Term 20 (EK1100-0018)^Term 28 (EL1859)^Channel 5^Input'}
	nv_3162_a_open_feedback AT %I* : BOOL;
	
	//Digital valve closed feedback
	//{attribute 'TcLinkTo' := 'TIID^Device 1 (EtherCAT)^Term 31 (EK1914)^Term 32 (EL1859)^Channel 11^Output'}
	nv_3110_a_closed_feedback AT %I* : BOOL;
	//{attribute 'TcLinkTo' := 'TIID^Device 1 (EtherCAT)^Term 31 (EK1914)^Term 32 (EL1859)^Channel 11^Output'}
	nv_3210_a_closed_feedback AT %I* : BOOL;
	//{attribute 'TcLinkTo' := 'TIID^Device 1 (EtherCAT)^Term 31 (EK1914)^Term 32 (EL1859)^Channel 11^Output'}
	nv_3310_a_closed_feedback AT %I* : BOOL;
	{attribute 'TcLinkTo' := 'TIID^Device 1 (EtherCAT)^Term 20 (EK1100-0018)^Term 29 (EL1859)^Channel 1^Input'}
	nv_3135_a_closed_feedback AT %I* : BOOL;
	{attribute 'TcLinkTo' := 'TIID^Device 1 (EtherCAT)^Term 20 (EK1100-0018)^Term 29 (EL1859)^Channel 2^Input'}
	nv_3235_a_closed_feedback AT %I* : BOOL;
	{attribute 'TcLinkTo' := 'TIID^Device 1 (EtherCAT)^Term 20 (EK1100-0018)^Term 29 (EL1859)^Channel 3^Input'}
	nv_3335_a_closed_feedback AT %I* : BOOL;
	{attribute 'TcLinkTo' := 'TIID^Device 1 (EtherCAT)^Term 20 (EK1100-0018)^Term 29 (EL1859)^Channel 4^Input'}
	nv_3372_a_closed_feedback AT %I* : BOOL;
	{attribute 'TcLinkTo' := 'TIID^Device 1 (EtherCAT)^Term 20 (EK1100-0018)^Term 29 (EL1859)^Channel 5^Input'}
	nv_3162_a_closed_feedback AT %I* : BOOL;
	

END_VAR

//---Field Instrumentation--------------------------------------------------------------------------------------------------

//Instantiate analog input function block
cpt_3144_a();
//Map values from the OPC GVL so that they can be written to from outside POU(IE from HMI)
cpt_3144_a.eu_max:=opc.popa_0081_cpt_3144_a_eu_max;
cpt_3144_a.eu_min:=opc.popa_0081_cpt_3144_a_eu_min;
cpt_3144_a.filter_factor:=opc.popa_0081_cpt_3144_a_filter_factor;
cpt_3144_a.raw_max:=opc.popa_0081_cpt_3144_a_raw_max;
cpt_3144_a.raw_min:=opc.popa_0081_cpt_3144_a_raw_min;
//Map the analog scaling function block raw input to the physical raw input variable
cpt_3144_a.raw_input := cpt_3144_a_raw_input;

//Instantiate analog input function block
cct_3120_a();
//Map values from the OPC GVL so that they can be written to from outside POU(IE from HMI)
cct_3120_a.eu_max:=opc.popa_0081_cct_3120_a_eu_max;
cct_3120_a.eu_min:=opc.popa_0081_cct_3120_a_eu_min;
cct_3120_a.filter_factor:=opc.popa_0081_cct_3120_a_filter_factor;
cct_3120_a.raw_max:=opc.popa_0081_cct_3120_a_raw_max;
cct_3120_a.raw_min:=opc.popa_0081_cct_3120_a_raw_min;
//Map the analog scaling function block raw input to the physical raw input variable
cct_3120_a.raw_input := cct_3120_a_raw_input;

//Instantiate analog input function block
cct_3220_a();
//Map values from the OPC GVL so that they can be written to from outside POU(IE from HMI)
cct_3220_a.eu_max:=opc.popa_0081_cct_3220_a_eu_max;
cct_3220_a.eu_min:=opc.popa_0081_cct_3220_a_eu_min;
cct_3220_a.filter_factor:=opc.popa_0081_cct_3220_a_filter_factor;
cct_3220_a.raw_max:=opc.popa_0081_cct_3220_a_raw_max;
cct_3220_a.raw_min:=opc.popa_0081_cct_3220_a_raw_min;
//Map the analog scaling function block raw input to the physical raw input variable
cct_3220_a.raw_input := cct_3220_a_raw_input;

//Instantiate analog input function block
cct_3320_a();
//Map values from the OPC GVL so that they can be written to from outside POU(IE from HMI)
cct_3320_a.eu_max:=opc.popa_0081_cct_3320_a_eu_max;
cct_3320_a.eu_min:=opc.popa_0081_cct_3320_a_eu_min;
cct_3320_a.filter_factor:=opc.popa_0081_cct_3320_a_filter_factor;
cct_3320_a.raw_max:=opc.popa_0081_cct_3320_a_raw_max;
cct_3320_a.raw_min:=opc.popa_0081_cct_3320_a_raw_min;
//Map the analog scaling function block raw input to the physical raw input variable
cct_3320_a.raw_input := cct_3320_a_raw_input;

//Instantiate analog input function block
cct_3142_a();
//Map values from the OPC GVL so that they can be written to from outside POU(IE from HMI)
cct_3142_a.eu_max:=opc.popa_0081_cct_3142_a_eu_max;
cct_3142_a.eu_min:=opc.popa_0081_cct_3142_a_eu_min;
cct_3142_a.filter_factor:=opc.popa_0081_cct_3142_a_filter_factor;
cct_3142_a.raw_max:=opc.popa_0081_cct_3142_a_raw_max;
cct_3142_a.raw_min:=opc.popa_0081_cct_3142_a_raw_min;
//Map the analog scaling function block raw input to the physical raw input variable
cct_3142_a.raw_input := cct_3142_a_raw_input;

//Instantiate analog input function block
cct_3242_a();
//Map values from the OPC GVL so that they can be written to from outside POU(IE from HMI)
cct_3242_a.eu_max:=opc.popa_0081_cct_3242_a_eu_max;
cct_3242_a.eu_min:=opc.popa_0081_cct_3242_a_eu_min;
cct_3242_a.filter_factor:=opc.popa_0081_cct_3242_a_filter_factor;
cct_3242_a.raw_max:=opc.popa_0081_cct_3242_a_raw_max;
cct_3242_a.raw_min:=opc.popa_0081_cct_3242_a_raw_min;
//Map the analog scaling function block raw input to the physical raw input variable
cct_3242_a.raw_input := cct_3242_a_raw_input;

//Instantiate analog input function block
cct_3342_a();
//Map values from the OPC GVL so that they can be written to from outside POU(IE from HMI)
cct_3342_a.eu_max:=opc.popa_0081_cct_3342_a_eu_max;
cct_3342_a.eu_min:=opc.popa_0081_cct_3342_a_eu_min;
cct_3342_a.filter_factor:=opc.popa_0081_cct_3342_a_filter_factor;
cct_3342_a.raw_max:=opc.popa_0081_cct_3342_a_raw_max;
cct_3342_a.raw_min:=opc.popa_0081_cct_3342_a_raw_min;
//Map the analog scaling function block raw input to the physical raw input variable
cct_3342_a.raw_input := cct_3342_a_raw_input;

//Instantiate analog input function block
ft_3122_a();
//Map values from the OPC GVL so that they can be written to from outside POU(IE from HMI)
ft_3122_a.eu_max:=500;//opc.popa_0081_ft_3122_a_eu_max;
ft_3122_a.eu_min:=opc.popa_0081_ft_3122_a_eu_min;
ft_3122_a.filter_factor:=opc.popa_0081_ft_3122_a_filter_factor;
ft_3122_a.raw_max:=opc.popa_0081_ft_3122_a_raw_max;
ft_3122_a.raw_min:=opc.popa_0081_ft_3122_a_raw_min;
//Map the analog scaling function block raw input to the physical raw input variable
ft_3122_a.raw_input := ft_3122_a_raw_input;

//Instantiate analog input function block
ft_3222_a();
//Map values from the OPC GVL so that they can be written to from outside POU(IE from HMI)
ft_3222_a.eu_max:=500;//opc.popa_0081_ft_3222_a_eu_max;
ft_3222_a.eu_min:=opc.popa_0081_ft_3222_a_eu_min;
ft_3222_a.filter_factor:=opc.popa_0081_ft_3222_a_filter_factor;
ft_3222_a.raw_max:=opc.popa_0081_ft_3222_a_raw_max;
ft_3222_a.raw_min:=opc.popa_0081_ft_3222_a_raw_min;
//Map the analog scaling function block raw input to the physical raw input variable
ft_3222_a.raw_input := ft_3222_a_raw_input;

//Instantiate analog input function block
ft_3322_a();
//Map values from the OPC GVL so that they can be written to from outside POU(IE from HMI)
ft_3322_a.eu_max:=500;//opc.popa_0081_ft_3322_a_eu_max;
ft_3322_a.eu_min:=opc.popa_0081_ft_3322_a_eu_min;
ft_3322_a.filter_factor:=opc.popa_0081_ft_3322_a_filter_factor;
ft_3322_a.raw_max:=opc.popa_0081_ft_3322_a_raw_max;
ft_3322_a.raw_min:=opc.popa_0081_ft_3322_a_raw_min;
//Map the analog scaling function block raw input to the physical raw input variable
ft_3322_a.raw_input := ft_3322_a_raw_input;

//Instantiate analog input function block
lt_3102_a();
//Map values from the OPC GVL so that they can be written to from outside POU(IE from HMI)
lt_3102_a.eu_max:=opc.popa_0081_lt_3102_a_eu_max;
lt_3102_a.eu_min:=opc.popa_0081_lt_3102_a_eu_min;
lt_3102_a.filter_factor:=opc.popa_0081_lt_3102_a_filter_factor;
lt_3102_a.raw_max:=opc.popa_0081_lt_3102_a_raw_max;
lt_3102_a.raw_min:=opc.popa_0081_lt_3102_a_raw_min;
//Map the analog scaling function block raw input to the physical raw input variable
lt_3102_a.raw_input := lt_3102_a_raw_input;

//Instantiate analog input function block
lt_3202_a();
//Map values from the OPC GVL so that they can be written to from outside POU(IE from HMI)
lt_3202_a.eu_max:=opc.popa_0081_lt_3202_a_eu_max;
lt_3202_a.eu_min:=opc.popa_0081_lt_3202_a_eu_min;
lt_3202_a.filter_factor:=opc.popa_0081_lt_3202_a_filter_factor;
lt_3202_a.raw_max:=opc.popa_0081_lt_3202_a_raw_max;
lt_3202_a.raw_min:=opc.popa_0081_lt_3202_a_raw_min;
//Map the analog scaling function block raw input to the physical raw input variable
lt_3202_a.raw_input := lt_3202_a_raw_input;

//Instantiate analog input function block
lt_3302_a();
//Map values from the OPC GVL so that they can be written to from outside POU(IE from HMI)
lt_3302_a.eu_max:=opc.popa_0081_lt_3302_a_eu_max;
lt_3302_a.eu_min:=opc.popa_0081_lt_3302_a_eu_min;
lt_3302_a.filter_factor:=opc.popa_0081_lt_3302_a_filter_factor;
lt_3302_a.raw_max:=opc.popa_0081_lt_3302_a_raw_max;
lt_3302_a.raw_min:=opc.popa_0081_lt_3302_a_raw_min;
//Map the analog scaling function block raw input to the physical raw input variable
lt_3302_a.raw_input := lt_3302_a_raw_input;

//Instantiate analog input function block
lt_3153_a();
//Map values from the OPC GVL so that they can be written to from outside POU(IE from HMI)
lt_3153_a.eu_max:=opc.popa_0081_lt_3153_a_eu_max;
lt_3153_a.eu_min:=opc.popa_0081_lt_3153_a_eu_min;
lt_3153_a.filter_factor:=opc.popa_0081_lt_3153_a_filter_factor;
lt_3153_a.raw_max:=opc.popa_0081_lt_3153_a_raw_max;
lt_3153_a.raw_min:=opc.popa_0081_lt_3153_a_raw_min;
//Map the analog scaling function block raw input to the physical raw input variable
lt_3153_a.raw_input := lt_3153_a_raw_input;

//Instantiate analog input function block
lt_3253_a();
//Map values from the OPC GVL so that they can be written to from outside POU(IE from HMI)
lt_3253_a.eu_max:=opc.popa_0081_lt_3253_a_eu_max;
lt_3253_a.eu_min:=opc.popa_0081_lt_3253_a_eu_min;
lt_3253_a.filter_factor:=opc.popa_0081_lt_3253_a_filter_factor;
lt_3253_a.raw_max:=opc.popa_0081_lt_3253_a_raw_max;
lt_3253_a.raw_min:=opc.popa_0081_lt_3253_a_raw_min;
//Map the analog scaling function block raw input to the physical raw input variable
lt_3253_a.raw_input := lt_3253_a_raw_input;

//Instantiate analog input function block
lt_3353_a();
//Map values from the OPC GVL so that they can be written to from outside POU(IE from HMI)
lt_3353_a.eu_max:=opc.popa_0081_lt_3353_a_eu_max;
lt_3353_a.eu_min:=opc.popa_0081_lt_3353_a_eu_min;
lt_3353_a.filter_factor:=opc.popa_0081_lt_3353_a_filter_factor;
lt_3353_a.raw_max:=opc.popa_0081_lt_3353_a_raw_max;
lt_3353_a.raw_min:=opc.popa_0081_lt_3353_a_raw_min;
//Map the analog scaling function block raw input to the physical raw input variable
lt_3353_a.raw_input := lt_3353_a_raw_input;

//Instantiate analog input function block
lt_3402_a();
//Map values from the OPC GVL so that they can be written to from outside POU(IE from HMI)
lt_3402_a.eu_max:=opc.popa_0091_lt_3402_a_eu_max;
lt_3402_a.eu_min:=opc.popa_0091_lt_3402_a_eu_min;
lt_3402_a.filter_factor:=opc.popa_0091_lt_3402_a_filter_factor;
lt_3402_a.raw_max:=opc.popa_0091_lt_3402_a_raw_max;
lt_3402_a.raw_min:=opc.popa_0091_lt_3402_a_raw_min;
//Map the analog scaling function block raw input to the physical raw input variable
lt_3402_a.raw_input := lt_3402_a_raw_input;

//Instantiate analog input function block
pt_3119_a();
//Map values from the OPC GVL so that they can be written to from outside POU(IE from HMI)
pt_3119_a.eu_max:=opc.popa_0081_pt_3119_a_eu_max;
pt_3119_a.eu_min:=opc.popa_0081_pt_3119_a_eu_min;
pt_3119_a.filter_factor:=opc.popa_0081_pt_3119_a_filter_factor;
pt_3119_a.raw_max:=opc.popa_0081_pt_3119_a_raw_max;
pt_3119_a.raw_min:=opc.popa_0081_pt_3119_a_raw_min;
//Map the analog scaling function block raw input to the physical raw input variable
pt_3119_a.raw_input := pt_3119_a_raw_input;

//Instantiate analog input function block
pt_3219_a();
//Map values from the OPC GVL so that they can be written to from outside POU(IE from HMI)
pt_3219_a.eu_max:=opc.popa_0081_pt_3219_a_eu_max;
pt_3219_a.eu_min:=opc.popa_0081_pt_3219_a_eu_min;
pt_3219_a.filter_factor:=opc.popa_0081_pt_3219_a_filter_factor;
pt_3219_a.raw_max:=opc.popa_0081_pt_3219_a_raw_max;
pt_3219_a.raw_min:=opc.popa_0081_pt_3219_a_raw_min;
//Map the analog scaling function block raw input to the physical raw input variable
pt_3219_a.raw_input := pt_3219_a_raw_input;

//Instantiate analog input function block
pt_3319_a();
//Map values from the OPC GVL so that they can be written to from outside POU(IE from HMI)
pt_3319_a.eu_max:=opc.popa_0081_pt_3319_a_eu_max;
pt_3319_a.eu_min:=opc.popa_0081_pt_3319_a_eu_min;
pt_3319_a.filter_factor:=opc.popa_0081_pt_3319_a_filter_factor;
pt_3319_a.raw_max:=opc.popa_0081_pt_3319_a_raw_max;
pt_3319_a.raw_min:=opc.popa_0081_pt_3319_a_raw_min;
//Map the analog scaling function block raw input to the physical raw input variable
pt_3319_a.raw_input := pt_3319_a_raw_input;

//Instantiate analog input function block
pt_3141_a();
//Map values from the OPC GVL so that they can be written to from outside POU(IE from HMI)
pt_3141_a.eu_max:=opc.popa_0081_pt_3141_a_eu_max;
pt_3141_a.eu_min:=opc.popa_0081_pt_3141_a_eu_min;
pt_3141_a.filter_factor:=opc.popa_0081_pt_3141_a_filter_factor;
pt_3141_a.raw_max:=opc.popa_0081_pt_3141_a_raw_max;
pt_3141_a.raw_min:=opc.popa_0081_pt_3141_a_raw_min;
//Map the analog scaling function block raw input to the physical raw input variable
pt_3141_a.raw_input := pt_3141_a_raw_input;

//Instantiate analog input function block
pt_3241_a();
//Map values from the OPC GVL so that they can be written to from outside POU(IE from HMI)
pt_3241_a.eu_max:=opc.popa_0081_pt_3241_a_eu_max;
pt_3241_a.eu_min:=opc.popa_0081_pt_3241_a_eu_min;
pt_3241_a.filter_factor:=opc.popa_0081_pt_3241_a_filter_factor;
pt_3241_a.raw_max:=opc.popa_0081_pt_3241_a_raw_max;
pt_3241_a.raw_min:=opc.popa_0081_pt_3241_a_raw_min;
//Map the analog scaling function block raw input to the physical raw input variable
pt_3241_a.raw_input := pt_3241_a_raw_input;

//Instantiate analog input function block
pt_3341_a();
//Map values from the OPC GVL so that they can be written to from outside POU(IE from HMI)
pt_3341_a.eu_max:=opc.popa_0081_pt_3341_a_eu_max;
pt_3341_a.eu_min:=opc.popa_0081_pt_3341_a_eu_min;
pt_3341_a.filter_factor:=opc.popa_0081_pt_3341_a_filter_factor;
pt_3341_a.raw_max:=opc.popa_0081_pt_3341_a_raw_max;
pt_3341_a.raw_min:=opc.popa_0081_pt_3341_a_raw_min;
//Map the analog scaling function block raw input to the physical raw input variable
pt_3341_a.raw_input := pt_3341_a_raw_input;

//Instantiate analog input function block
pt_3428_a();
//Map values from the OPC GVL so that they can be written to from outside POU(IE from HMI)
pt_3428_a.eu_max:=opc.popa_0091_pt_3428_a_eu_max;
pt_3428_a.eu_min:=opc.popa_0091_pt_3428_a_eu_min;
pt_3428_a.filter_factor:=opc.popa_0091_pt_3428_a_filter_factor;
pt_3428_a.raw_max:=opc.popa_0091_pt_3428_a_raw_max;
pt_3428_a.raw_min:=opc.popa_0091_pt_3428_a_raw_min;
//Map the analog scaling function block raw input to the physical raw input variable
pt_3428_a.raw_input := pt_3428_a_raw_input;

//Instantiate analog input function block
pt_3414_a();
//Map values from the OPC GVL so that they can be written to from outside POU(IE from HMI)
pt_3414_a.eu_max:=opc.popa_0091_pt_3414_a_eu_max;
pt_3414_a.eu_min:=opc.popa_0091_pt_3414_a_eu_min;
pt_3414_a.filter_factor:=opc.popa_0091_pt_3414_a_filter_factor;
pt_3414_a.raw_max:=opc.popa_0091_pt_3414_a_raw_max;
pt_3414_a.raw_min:=opc.popa_0091_pt_3414_a_raw_min;
//Map the analog scaling function block raw input to the physical raw input variable
pt_3414_a.raw_input := pt_3414_a_raw_input;

//Instantiate analog input function block
tt_3118_a();
//Map values from the OPC GVL so that they can be written to from outside POU(IE from HMI)
tt_3118_a.eu_max:=opc.popa_0081_tt_3118_a_eu_max;
tt_3118_a.eu_min:=opc.popa_0081_tt_3118_a_eu_min;
tt_3118_a.filter_factor:=opc.popa_0081_tt_3118_a_filter_factor;
tt_3118_a.raw_max:=opc.popa_0081_tt_3118_a_raw_max;
tt_3118_a.raw_min:=opc.popa_0081_tt_3118_a_raw_min;
//Map the analog scaling function block raw input to the physical raw input variable
tt_3118_a.raw_input := tt_3118_a_raw_input;

//Instantiate analog input function block
tt_3218_a();
//Map values from the OPC GVL so that they can be written to from outside POU(IE from HMI)
tt_3218_a.eu_max:=opc.popa_0081_tt_3218_a_eu_max;
tt_3218_a.eu_min:=opc.popa_0081_tt_3218_a_eu_min;
tt_3218_a.filter_factor:=opc.popa_0081_tt_3218_a_filter_factor;
tt_3218_a.raw_max:=opc.popa_0081_tt_3218_a_raw_max;
tt_3218_a.raw_min:=opc.popa_0081_tt_3218_a_raw_min;
//Map the analog scaling function block raw input to the physical raw input variable
tt_3218_a.raw_input := tt_3218_a_raw_input;

//Instantiate analog input function block
tt_3318_a();
//Map values from the OPC GVL so that they can be written to from outside POU(IE from HMI)
tt_3318_a.eu_max:=opc.popa_0081_tt_3318_a_eu_max;
tt_3318_a.eu_min:=opc.popa_0081_tt_3318_a_eu_min;
tt_3318_a.filter_factor:=opc.popa_0081_tt_3318_a_filter_factor;
tt_3318_a.raw_max:=opc.popa_0081_tt_3318_a_raw_max;
tt_3318_a.raw_min:=opc.popa_0081_tt_3318_a_raw_min;
//Map the analog scaling function block raw input to the physical raw input variable
tt_3318_a.raw_input := tt_3318_a_raw_input;

//Instantiate analog input function block
tt_3140_a();
//Map values from the OPC GVL so that they can be written to from outside POU(IE from HMI)
tt_3140_a.eu_max:=opc.popa_0081_tt_3140_a_eu_max;
tt_3140_a.eu_min:=opc.popa_0081_tt_3140_a_eu_min;
tt_3140_a.filter_factor:=opc.popa_0081_tt_3140_a_filter_factor;
tt_3140_a.raw_max:=opc.popa_0081_tt_3140_a_raw_max;
tt_3140_a.raw_min:=opc.popa_0081_tt_3140_a_raw_min;
//Map the analog scaling function block raw input to the physical raw input variable
tt_3140_a.raw_input := tt_3140_a_raw_input;

//Instantiate analog input function block
tt_3240_a();
//Map values from the OPC GVL so that they can be written to from outside POU(IE from HMI)
tt_3240_a.eu_max:=opc.popa_0081_tt_3240_a_eu_max;
tt_3240_a.eu_min:=opc.popa_0081_tt_3240_a_eu_min;
tt_3240_a.filter_factor:=opc.popa_0081_tt_3240_a_filter_factor;
tt_3240_a.raw_max:=opc.popa_0081_tt_3240_a_raw_max;
tt_3240_a.raw_min:=opc.popa_0081_tt_3240_a_raw_min;
//Map the analog scaling function block raw input to the physical raw input variable
tt_3240_a.raw_input := tt_3240_a_raw_input;

//Instantiate analog input function block
tt_3340_a();
//Map values from the OPC GVL so that they can be written to from outside POU(IE from HMI)
tt_3340_a.eu_max:=opc.popa_0081_tt_3340_a_eu_max;
tt_3340_a.eu_min:=opc.popa_0081_tt_3340_a_eu_min;
tt_3340_a.filter_factor:=opc.popa_0081_tt_3340_a_filter_factor;
tt_3340_a.raw_max:=opc.popa_0081_tt_3340_a_raw_max;
tt_3340_a.raw_min:=opc.popa_0081_tt_3340_a_raw_min;
//Map the analog scaling function block raw input to the physical raw input variable
tt_3340_a.raw_input := tt_3340_a_raw_input;

//Instantiate analog input function block
tt_3432_a();
//Map values from the OPC GVL so that they can be written to from outside POU(IE from HMI)
tt_3432_a.eu_max:=opc.popa_0091_tt_3432_a_eu_max;
tt_3432_a.eu_min:=opc.popa_0091_tt_3432_a_eu_min;
tt_3432_a.filter_factor:=opc.popa_0091_tt_3432_a_filter_factor;
tt_3432_a.raw_max:=opc.popa_0091_tt_3432_a_raw_max;
tt_3432_a.raw_min:=opc.popa_0091_tt_3432_a_raw_min;
//Map the analog scaling function block raw input to the physical raw input variable
tt_3432_a.raw_input := tt_3432_a_raw_input;

//---Pumps---------------------------------------------------------------------------------------------------------------------------------



//Instantiate u_3112_a speed feedback analog input function block
u_3112_a_speed_feedback();
//Map values from the OPC GVL so that they can be written to from outside POU(IE from HMI)
u_3112_a_speed_feedback.eu_max:=60;
u_3112_a_speed_feedback.eu_min:=0;
u_3112_a_speed_feedback.filter_factor:=opc.popa_0081_u_3112_a_speed_feedback_filter_factor;
u_3112_a_speed_feedback.raw_max:=opc.popa_0081_u_3112_a_speed_feedback_raw_max;
u_3112_a_speed_feedback.raw_min:=opc.popa_0081_u_3112_a_speed_feedback_raw_min;
//Map the analog scaling function block raw input to the physical raw input variable
u_3112_a_speed_feedback.raw_input := u_3112_a_speed_feedback_raw_input;





//--------------------------------------------------------------------------------------------------------------


//Instantiate Example analog input function block
u_3212_a_speed_feedback();
//Map values from the OPC GVL so that they can be written to from outside POU(IE from HMI)
u_3212_a_speed_feedback.eu_max:=60;
u_3212_a_speed_feedback.eu_min:=0;
u_3212_a_speed_feedback.filter_factor:=opc.popa_0081_u_3212_a_speed_feedback_filter_factor;
u_3212_a_speed_feedback.raw_max:=opc.popa_0081_u_3212_a_speed_feedback_raw_max;
u_3212_a_speed_feedback.raw_min:=opc.popa_0081_u_3212_a_speed_feedback_raw_min;
//Map the analog scaling function block raw input to the physical raw input variable
u_3212_a_speed_feedback.raw_input := u_3212_a_speed_feedback_raw_input;

//--------------------------------------------------------------------------------------------------------------


//Instantiate Example analog input function block
u_3312_a_speed_feedback();
//Map values from the OPC GVL so that they can be written to from outside POU(IE from HMI)
u_3312_a_speed_feedback.eu_max:=60;
u_3312_a_speed_feedback.eu_min:=0;
u_3312_a_speed_feedback.filter_factor:=opc.popa_0081_u_3312_a_speed_feedback_filter_factor;
u_3312_a_speed_feedback.raw_max:=opc.popa_0081_u_3312_a_speed_feedback_raw_max;
u_3312_a_speed_feedback.raw_min:=opc.popa_0081_u_3312_a_speed_feedback_raw_min;
//Map the analog scaling function block raw input to the physical raw input variable
u_3312_a_speed_feedback.raw_input := u_3312_a_speed_feedback_raw_input;

//--------------------------------------------------------------------------------------------------------------


//Instantiate Example analog input function block
u_3160_a_speed_feedback();
//Map values from the OPC GVL so that they can be written to from outside POU(IE from HMI)
u_3160_a_speed_feedback.eu_max:=60;
u_3160_a_speed_feedback.eu_min:=0;
u_3160_a_speed_feedback.filter_factor:=opc.popa_0081_u_3160_a_speed_feedback_filter_factor;
u_3160_a_speed_feedback.raw_max:=opc.popa_0081_u_3160_a_speed_feedback_raw_max;
u_3160_a_speed_feedback.raw_min:=opc.popa_0081_u_3160_a_speed_feedback_raw_min;
//Map the analog scaling function block raw input to the physical raw input variable
u_3160_a_speed_feedback.raw_input := u_3160_a_speed_feedback_raw_input;

//--------------------------------------------------------------------------------------------------------------


//Instantiate Example analog input function block
u_3260_a_speed_feedback();
//Map values from the OPC GVL so that they can be written to from outside POU(IE from HMI)
u_3260_a_speed_feedback.eu_max:=60;
u_3260_a_speed_feedback.eu_min:=0;
u_3260_a_speed_feedback.filter_factor:=opc.popa_0081_u_3260_a_speed_feedback_filter_factor;
u_3260_a_speed_feedback.raw_max:=opc.popa_0081_u_3260_a_speed_feedback_raw_max;
u_3260_a_speed_feedback.raw_min:=opc.popa_0081_u_3260_a_speed_feedback_raw_min;
//Map the analog scaling function block raw input to the physical raw input variable
u_3260_a_speed_feedback.raw_input := u_3260_a_speed_feedback_raw_input;

//--------------------------------------------------------------------------------------------------------------


//Instantiate Example analog input function block
u_3360_a_speed_feedback();
//Map values from the OPC GVL so that they can be written to from outside POU(IE from HMI)
u_3360_a_speed_feedback.eu_max:=60;
u_3360_a_speed_feedback.eu_min:=0;
u_3360_a_speed_feedback.filter_factor:=opc.popa_0081_u_3360_a_speed_feedback_filter_factor;
u_3360_a_speed_feedback.raw_max:=opc.popa_0081_u_3360_a_speed_feedback_raw_max;
u_3360_a_speed_feedback.raw_min:=opc.popa_0081_u_3360_a_speed_feedback_raw_min;
//Map the analog scaling function block raw input to the physical raw input variable
u_3360_a_speed_feedback.raw_input := u_3360_a_speed_feedback_raw_input;

//--------------------------------------------------------------------------------------------------------------


//Instantiate Example analog input function block
u_3370_a_speed_feedback();
//Map values from the OPC GVL so that they can be written to from outside POU(IE from HMI)
u_3370_a_speed_feedback.eu_max:=60;
u_3370_a_speed_feedback.eu_min:=0;
u_3370_a_speed_feedback.filter_factor:=opc.popa_0081_u_3370_a_speed_feedback_filter_factor;
u_3370_a_speed_feedback.raw_max:=opc.popa_0081_u_3370_a_speed_feedback_raw_max;
u_3370_a_speed_feedback.raw_min:=opc.popa_0081_u_3370_a_speed_feedback_raw_min;
//Map the analog scaling function block raw input to the physical raw input variable
u_3370_a_speed_feedback.raw_input := u_3370_a_speed_feedback_raw_input;

//--------------------------------------------------------------------------------------------------------------


//Instantiate Example analog input function block
u_3405_a_speed_feedback();
//Map values from the OPC GVL so that they can be written to from outside POU(IE from HMI)
u_3405_a_speed_feedback.eu_max:=60;
u_3405_a_speed_feedback.eu_min:=0;
u_3405_a_speed_feedback.filter_factor:=opc.popa_0091_u_3405_a_speed_feedback_filter_factor;
u_3405_a_speed_feedback.raw_max:=opc.popa_0091_u_3405_a_speed_feedback_raw_max;
u_3405_a_speed_feedback.raw_min:=opc.popa_0091_u_3405_a_speed_feedback_raw_min;
//Map the analog scaling function block raw input to the physical raw input variable
u_3405_a_speed_feedback.raw_input := u_3405_a_speed_feedback_raw_input;


//---Valves----------------------------------------------------------------------------------------------------------------------------------------------

//Instantiate av_3148 analog input function block----------------------------------------------------------------------------
av_3148_a_position_feedback();
//Map values from the OPC GVL so that they can be written to from outside POU(IE from HMI)
av_3148_a_position_feedback.eu_max:=100;
av_3148_a_position_feedback.eu_min:=0;
av_3148_a_position_feedback.filter_factor:=opc.popa_0081_av_3148_a_position_feedback_filter_factor;
av_3148_a_position_feedback.raw_max:=opc.popa_0081_av_3148_a_position_feedback_raw_max;
av_3148_a_position_feedback.raw_min:=opc.popa_0081_av_3148_a_position_feedback_raw_min;
//Map the analog scaling function block raw input to the physical raw input variable
av_3148_a_position_feedback.raw_input := av_3148_a_position_feedback_raw_input;




//Instantiate av_3248 analog input function block-----------------------------------------------------------------
av_3248_a_position_feedback();
//Map values from the OPC GVL so that they can be written to from outside POU(IE from HMI)
av_3248_a_position_feedback.eu_max:=100;
av_3248_a_position_feedback.eu_min:=0;
av_3248_a_position_feedback.filter_factor:=opc.popa_0081_av_3248_a_position_feedback_filter_factor;
av_3248_a_position_feedback.raw_max:=opc.popa_0081_av_3248_a_position_feedback_raw_max;
av_3248_a_position_feedback.raw_min:=opc.popa_0081_av_3248_a_position_feedback_raw_min;
//Map the analog scaling function block raw input to the physical raw input variable
av_3248_a_position_feedback.raw_input := av_3248_a_position_feedback_raw_input;




//Instantiate av_3348 analog input function block----------------------------------------------------------------------
av_3348_a_position_feedback();
//Map values from the OPC GVL so that they can be written to from outside POU(IE from HMI)
av_3348_a_position_feedback.eu_max:=100;
av_3348_a_position_feedback.eu_min:=0;
av_3348_a_position_feedback.filter_factor:=opc.popa_0081_av_3348_a_position_feedback_filter_factor;
av_3348_a_position_feedback.raw_max:=opc.popa_0081_av_3348_a_position_feedback_raw_max;
av_3348_a_position_feedback.raw_min:=opc.popa_0081_av_3348_a_position_feedback_raw_min;
//Map the analog scaling function block raw input to the physical raw input variable
av_3348_a_position_feedback.raw_input := av_3348_a_position_feedback_raw_input;

END_PROGRAM

// ---- POUs/manual_mode.TcPOU
PROGRAM manual_mode
VAR
	//manual_mode: BOOL;
	
	u_3112_hmi_start_request: BOOL;
	u_3112_manual_request: BOOL;
	u_3112_hmi_speed_request: REAL;
	u_3112_manual_speed_request: REAL;
	u_3112_hmi_stop_request: BOOL;
	
	u_3212_hmi_start_request: BOOL;
	u_3212_manual_request: BOOL;
	u_3212_hmi_speed_request: REAL;
	u_3212_manual_speed_request: REAL;
	u_3212_hmi_stop_request: BOOL;

	u_3312_hmi_start_request: BOOL;
	u_3312_manual_request: BOOL;
	u_3312_hmi_speed_request: REAL;
	u_3312_manual_speed_request: REAL;
	u_3312_hmi_stop_request: BOOL;
	
	u_3405_hmi_start_request: BOOL;
	u_3405_manual_request: BOOL;
	u_3405_hmi_speed_request: REAL;
	u_3405_manual_speed_request: REAL;
	u_3405_hmi_stop_request: BOOL;
	
	u_3160_hmi_start_request: BOOL;
	u_3160_manual_request: BOOL;
	u_3160_hmi_speed_request: REAL;
	u_3160_manual_speed_request: REAL;
	u_3160_hmi_stop_request: BOOL;
	
	u_3260_hmi_start_request: BOOL;
	u_3260_manual_request: BOOL;
	u_3260_hmi_speed_request: REAL;
	u_3260_manual_speed_request: REAL;
	u_3260_hmi_stop_request: BOOL;
	
	u_3360_hmi_start_request: BOOL;
	u_3360_manual_request: BOOL;
	u_3360_hmi_speed_request: REAL;
	u_3360_manual_speed_request: REAL;
	u_3360_hmi_stop_request: BOOL;
	
	nv_3110_hmi_open_request: BOOL;
	nv_3110_hmi_close_request: BOOL;
	nv_3110_manual_request: BOOL;
	
	nv_3210_hmi_open_request: BOOL;
	nv_3210_hmi_close_request: BOOL;
	nv_3210_manual_request: BOOL;
	
	nv_3310_hmi_open_request: BOOL;
	nv_3310_hmi_close_request: BOOL;
	nv_3310_manual_request: BOOL;
	
	nv_3135_hmi_open_request: BOOL;
	nv_3135_hmi_close_request: BOOL;
	nv_3135_manual_request: BOOL;
	
	nv_3235_hmi_open_request: BOOL;
	nv_3235_hmi_close_request: BOOL;
	nv_3235_manual_request: BOOL;
	
	nv_3335_hmi_open_request: BOOL;
	nv_3335_hmi_close_request: BOOL;
	nv_3335_manual_request: BOOL;
	
	nv_3372_hmi_open_request: BOOL;
	nv_3372_hmi_close_request: BOOL;
	nv_3372_manual_request: BOOL;
	u_3370_hmi_start_request: BOOL;
	u_3370_manual_request: BOOL;
	u_3370_hmi_stop_request: BOOL;
	u_3370_hmi_speed_request: INT;
	u_3370_manual_speed_request: INT;
	nv_3162_hmi_open_request: BOOL;
	nv_3162_manual_request: BOOL;
	nv_3162_hmi_close_request: BOOL;
END_VAR

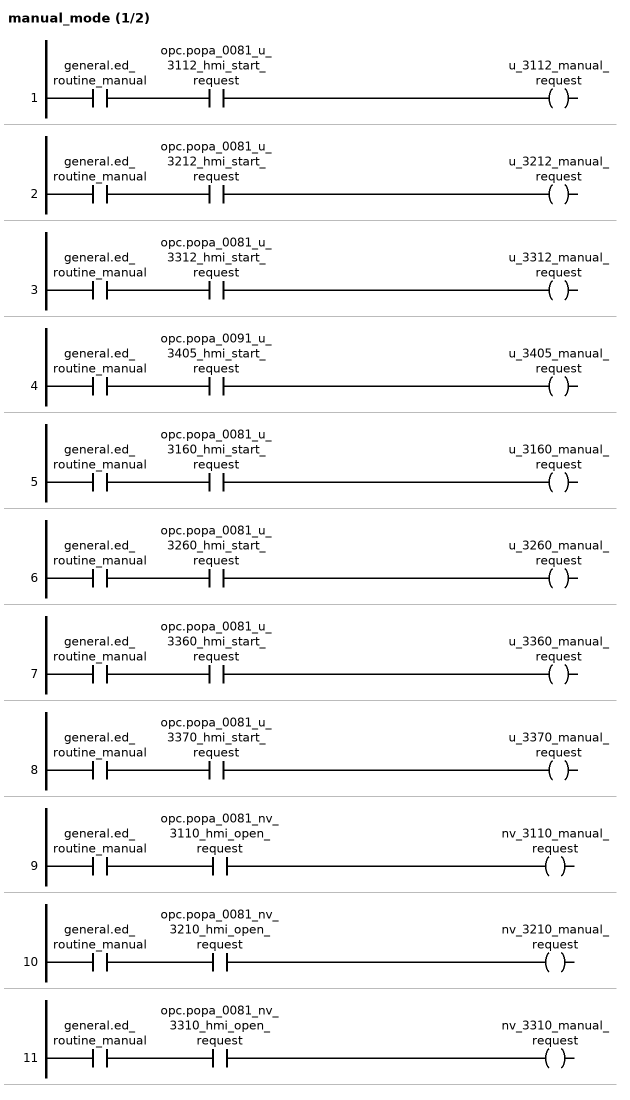
// NETWORK 1
u_3112_manual_request := general.ed_routine_manual AND opc.popa_0081_u_3112_hmi_start_request;

// NETWORK 2
u_3212_manual_request := general.ed_routine_manual AND opc.popa_0081_u_3212_hmi_start_request;

// NETWORK 3
u_3312_manual_request := general.ed_routine_manual AND opc.popa_0081_u_3312_hmi_start_request;

// NETWORK 4
u_3405_manual_request := general.ed_routine_manual AND opc.popa_0091_u_3405_hmi_start_request;

// NETWORK 5
u_3160_manual_request := general.ed_routine_manual AND opc.popa_0081_u_3160_hmi_start_request;

// NETWORK 6
u_3260_manual_request := general.ed_routine_manual AND opc.popa_0081_u_3260_hmi_start_request;

// NETWORK 7
u_3360_manual_request := general.ed_routine_manual AND opc.popa_0081_u_3360_hmi_start_request;

// NETWORK 8
u_3370_manual_request := general.ed_routine_manual AND opc.popa_0081_u_3370_hmi_start_request;

// NETWORK 9
nv_3110_manual_request := general.ed_routine_manual AND opc.popa_0081_nv_3110_hmi_open_request;

// NETWORK 10
nv_3210_manual_request := general.ed_routine_manual AND opc.popa_0081_nv_3210_hmi_open_request;

// NETWORK 11
nv_3310_manual_request := general.ed_routine_manual AND opc.popa_0081_nv_3310_hmi_open_request;

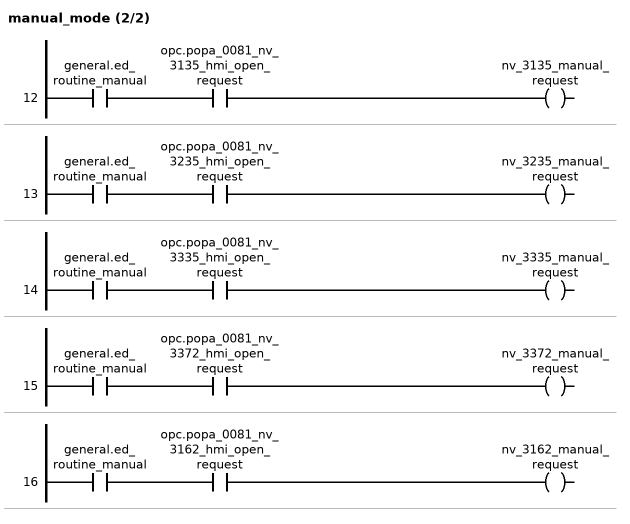
// NETWORK 12
nv_3135_manual_request := general.ed_routine_manual AND opc.popa_0081_nv_3135_hmi_open_request;

// NETWORK 13
nv_3235_manual_request := general.ed_routine_manual AND opc.popa_0081_nv_3235_hmi_open_request;

// NETWORK 14
nv_3335_manual_request := general.ed_routine_manual AND opc.popa_0081_nv_3335_hmi_open_request;

// NETWORK 15
nv_3372_manual_request := general.ed_routine_manual AND opc.popa_0081_nv_3372_hmi_open_request;

// NETWORK 16
nv_3162_manual_request := general.ed_routine_manual AND opc.popa_0081_nv_3162_hmi_open_request;

END_PROGRAM

// ---- POUs/interlocks.TcPOU
PROGRAM interlocks
VAR PERSISTENT
	nv_3110_open: BOOL;
	alm_lt_3012_low: BOOL;
	intlk_u3112: BOOL;
	nv_3210_open: BOOL;
	nv_3310_open: BOOL;
	intlk_u3212: BOOL;
	intlk_u3312: BOOL;
	alm_lt_3102_low: BOOL;
	alm_lt_3202_low: BOOL;
	alm_lt_3302_low: BOOL;
	alm_lt_3153_low: BOOL;
	intlk_u3160: BOOL;
	alm_lt_3253_low: BOOL;
	intlk_u3260: BOOL;
	alm_lt_3353_low: BOOL;
	intlk_u3360: BOOL;
	nv_3372_open: BOOL;
	intlk_u3370: BOOL;
	alm_lt_3402_low: BOOL;
	nv_3135_open: BOOL;
	nv_3235_open: BOOL;
	nv_3335: BOOL;
	nv_3335_open: BOOL;
	intlk_nv3110: BOOL;
	u_3112_running: BOOL;
END_VAR

VAR
	intlk_nv3210: BOOL;
	u_3212_running: BOOL;
	intlk_nv3310: BOOL;
	u_3312_running: BOOL;
	u_3112_intlk: BOOL;
	nv_3110_intlk: BOOL;
	u_3212_intlk: BOOL;
	nv_3210_intlk: BOOL;
	u_3312_intlk: BOOL;
	nv_3310_intlk: BOOL;
	u_3160_intlk: BOOL;
	u_3260_intlk: BOOL;
	u_3360_intlk: BOOL;
	u_3370_intlk: BOOL;
	u_3405_intlk: BOOL;
END_VAR

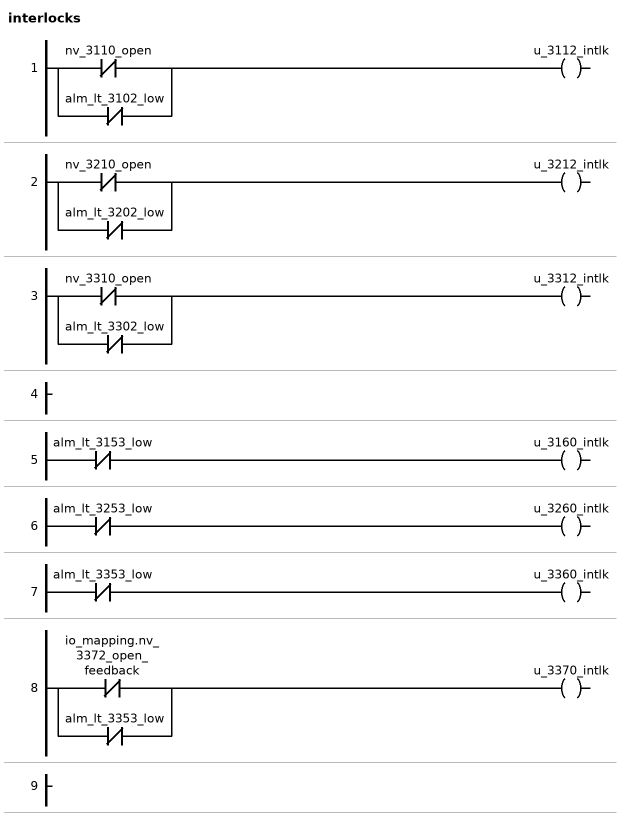
// NETWORK 1
u_3112_intlk := NOT nv_3110_open OR NOT alm_lt_3102_low;

// NETWORK 2
u_3212_intlk := NOT nv_3210_open OR NOT alm_lt_3202_low;

// NETWORK 3
u_3312_intlk := NOT nv_3310_open OR NOT alm_lt_3302_low;

// NETWORK 4

// NETWORK 5
u_3160_intlk := NOT alm_lt_3153_low;

// NETWORK 6
u_3260_intlk := NOT alm_lt_3253_low;

// NETWORK 7
u_3360_intlk := NOT alm_lt_3353_low;

// NETWORK 8
u_3370_intlk := NOT io_mapping.nv_3372_open_feedback OR NOT alm_lt_3353_low;

// NETWORK 9

END_PROGRAM

// ---- POUs/maint_mode.TcPOU
PROGRAM maint_mode
VAR
	maint_mode: BOOL;
	
	u_3112_a_hmi_start_request: BOOL;
	u_3112_a_maint_request: BOOL;
	u_3112_a_hmi_speed_request: REAL;
	u_3112_a_maint_speed_request: REAL;
	u_3112_a_hmi_stop_request: BOOL;
	
	u_3212_a_hmi_start_request: BOOL;
	u_3212_a_maint_request: BOOL;
	u_3212_a_hmi_speed_request: REAL;
	u_3212_a_maint_speed_request: REAL;
	u_3212_a_hmi_stop_request: BOOL;

	u_3312_a_hmi_start_request: BOOL;
	u_3312_a_maint_request: BOOL;
	u_3312_a_hmi_speed_request: REAL;
	u_3312_a_maint_speed_request: REAL;
	u_3312_a_hmi_stop_request: BOOL;
	
	u_3405_a_hmi_start_request: BOOL;
	u_3405_a_maint_request: BOOL;
	u_3405_a_hmi_speed_request: REAL;
	u_3405_a_maint_speed_request: REAL;
	u_3405_a_hmi_stop_request: BOOL;
	
	u_3160_a_hmi_start_request: BOOL;
	u_3160_a_maint_request: BOOL;
	u_3160_a_hmi_speed_request: REAL;
	u_3160_a_maint_speed_request: REAL;
	u_3160_a_hmi_stop_request: BOOL;
	
	u_3260_a_hmi_start_request: BOOL;
	u_3260_a_maint_request: BOOL;
	u_3260_a_hmi_speed_request: REAL;
	u_3260_a_maint_speed_request: REAL;
	u_3260_a_hmi_stop_request: BOOL;
	
	u_3360_a_hmi_start_request: BOOL;
	u_3360_a_maint_request: BOOL;
	u_3360_a_hmi_speed_request: REAL;
	u_3360_a_maint_speed_request: REAL;
	u_3360_a_hmi_stop_request: BOOL;
	
	nv_3110_a_hmi_open_request: BOOL;
	nv_3110_a_hmi_close_request: BOOL;
	nv_3110_a_maint_request: BOOL;
	
	nv_3210_a_hmi_open_request: BOOL;
	nv_3210_a_hmi_close_request: BOOL;
	nv_3210_a_maint_request: BOOL;
	
	nv_3310_a_hmi_open_request: BOOL;
	nv_3310_a_hmi_close_request: BOOL;
	nv_3310_a_maint_request: BOOL;
	
	nv_3135_a_hmi_open_request: BOOL;
	nv_3135_a_hmi_close_request: BOOL;
	nv_3135_a_maint_request: BOOL;
	
	nv_3235_a_hmi_open_request: BOOL;
	nv_3235_a_hmi_close_request: BOOL;
	nv_3235_a_maint_request: BOOL;
	
	nv_3335_a_hmi_open_request: BOOL;
	nv_3335_a_hmi_close_request: BOOL;
	nv_3335_a_maint_request: BOOL;
	
	nv_3372_a_hmi_open_request: BOOL;
	nv_3372_a_hmi_close_request: BOOL;
	nv_3372_a_maint_request: BOOL;
	u_3370_a_hmi_start_request: BOOL;
	u_3370_a_maint_request: BOOL;
	u_3370_a_hmi_stop_request: BOOL;
	u_3370_a_hmi_speed_request: REAL;
	u_3370_a_maint_speed_request: REAL;
	nv_3162_a_hmi_open_request: BOOL;
	nv_3162_a_maint_request: BOOL;
	nv_3162_a_hmi_close_request: BOOL;
END_VAR

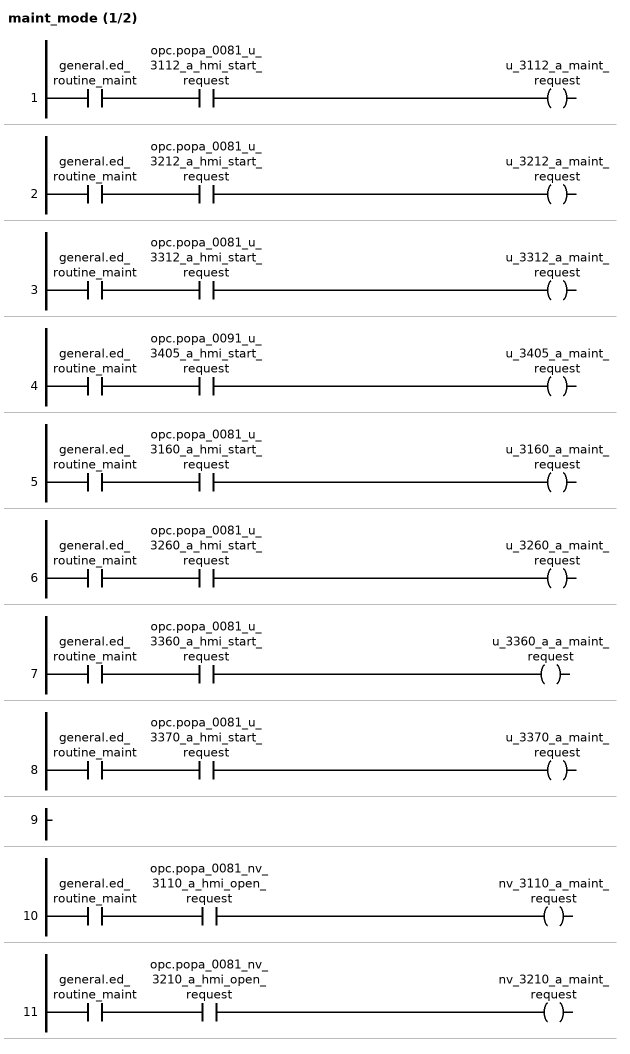
// NETWORK 1
u_3112_a_maint_request := general.ed_routine_maint AND opc.popa_0081_u_3112_a_hmi_start_request;

// NETWORK 2
u_3212_a_maint_request := general.ed_routine_maint AND opc.popa_0081_u_3212_a_hmi_start_request;

// NETWORK 3
u_3312_a_maint_request := general.ed_routine_maint AND opc.popa_0081_u_3312_a_hmi_start_request;

// NETWORK 4
u_3405_a_maint_request := general.ed_routine_maint AND opc.popa_0091_u_3405_a_hmi_start_request;

// NETWORK 5
u_3160_a_maint_request := general.ed_routine_maint AND opc.popa_0081_u_3160_a_hmi_start_request;

// NETWORK 6
u_3260_a_maint_request := general.ed_routine_maint AND opc.popa_0081_u_3260_a_hmi_start_request;

// NETWORK 7
u_3360_a_a_maint_request := general.ed_routine_maint AND opc.popa_0081_u_3360_a_hmi_start_request;

// NETWORK 8
u_3370_a_maint_request := general.ed_routine_maint AND opc.popa_0081_u_3370_a_hmi_start_request;

// NETWORK 9

// NETWORK 10
nv_3110_a_maint_request := general.ed_routine_maint AND opc.popa_0081_nv_3110_a_hmi_open_request;

// NETWORK 11
nv_3210_a_maint_request := general.ed_routine_maint AND opc.popa_0081_nv_3210_a_hmi_open_request;

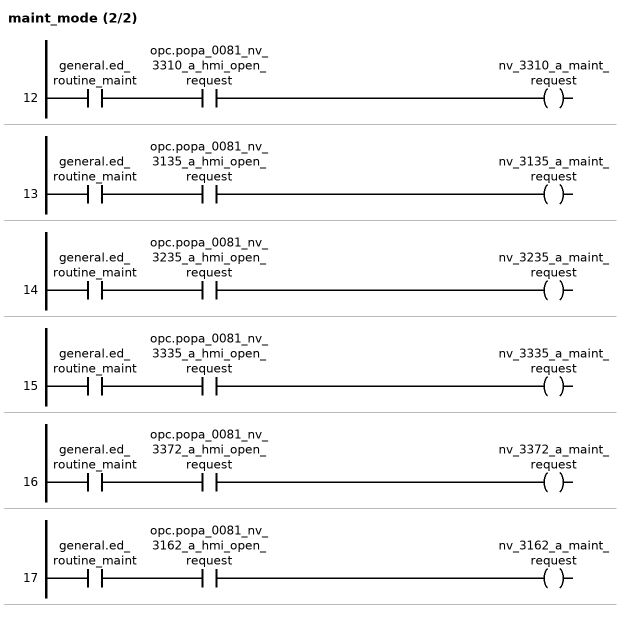
// NETWORK 12
nv_3310_a_maint_request := general.ed_routine_maint AND opc.popa_0081_nv_3310_a_hmi_open_request;

// NETWORK 13
nv_3135_a_maint_request := general.ed_routine_maint AND opc.popa_0081_nv_3135_a_hmi_open_request;

// NETWORK 14
nv_3235_a_maint_request := general.ed_routine_maint AND opc.popa_0081_nv_3235_a_hmi_open_request;

// NETWORK 15
nv_3335_a_maint_request := general.ed_routine_maint AND opc.popa_0081_nv_3335_a_hmi_open_request;

// NETWORK 16
nv_3372_a_maint_request := general.ed_routine_maint AND opc.popa_0081_nv_3372_a_hmi_open_request;

// NETWORK 17
nv_3162_a_maint_request := general.ed_routine_maint AND opc.popa_0081_nv_3162_a_hmi_open_request;

END_PROGRAM

// ---- POUs/stopping_mode.TcPOU
PROGRAM stopping_mode
VAR
	ed_routine_stopping_idle: BOOL;
	stack_power_enabled: BOOL;
	RECTIFIER_OUTPUT_OFF: BOOL;// ADD LOGIC FOR MONITORING RECTIFIER OUTPUT - USE CT? VERIFY PS DOES NOT MOVE CURRENT WHEN POWERED OFF
	u_3112_a_stop_request: BOOL;
	u_3212_a_stop_request: BOOL;
	u_3312_a_stop_request: BOOL;
	u_3405_a_stop_request: BOOL;
	u_3160_a_stop_request: BOOL
;
	u_3260_a_stop_request: BOOL;
	u_3360_a_stop_request: BOOL;
	u_3370_a_stop_request: BOOL;
	u_3112_a_run_feedback: BOOL;
	u_3212_a_run_feedback: BOOL;
	u_3312_a_run_feedback: BOOL;
	u_3405_a_run_feedback: BOOL;
	u_3160_a_run_feedback: BOOL;
	u_3260_a_run_feedback: BOOL;
	u_3360_a_run_feedback: BOOL;
	u_3370_a_run_feedback: BOOL;
	
	nv_3110_a_stop_request:BOOL;
	av_3248_a_stop_request: BOOL;
	av_3148_a_stop_request: BOOL;
	nv_3335_a_stop_request: BOOL;
	nv_3235_a_stop_request: BOOL;
	nv_3135_a_stop_request: BOOL;
	nv_3310_a_stop_request: BOOL;
	nv_3210_a_stop_request: BOOL;
	ed_routine_stop_mode: BOOL;
	redox_doser_stop_request: BOOL;
	nv_3335_a_position_request: INT;
	av_3148_a_position_request: INT;
	av_3248_a_position_request: INT;
	ed_pumps_stopped: BOOL;

	nv_3335_a_position_feedback: INT;
	nv_3335_a_recycle_position: BOOL;
	av_3148_a_position_feedback: INT;
	av_3148_a_recycle_position: BOOL;
	av_3248_a_recycle_position: BOOL;
	ed_valves_stopped: BOOL;
	ed_stopped: BOOL;
	av_3348_a_position_request: INT;
	nv_3372_a_stop_request: BOOL;
	av_3348_a_position_feedback: INT;
	av_3348_a_recycle_position: BOOL;
	nv_3335_a_closed_feedback: BOOL;
	nv_3372_a_closed_feedback: BOOL;
	nv_3162_a_stop_request: BOOL;
	ed_critical_stop: BOOL;
	tmr_stop_pump_delay: TON;
	tmr_stop_pump_delay_pt: TIME := T#10S;
	tmr_stop_pump_delay_et: TIME;
	test_ramp: ramp;
	eng_test: BOOL;
	test_ramp_start_val: REAL;
	test_ramp_end_val: REAL;
	test_ramp_duration: INT;
END_VAR
VAR // added by the converter: edge detectors and wires of the graphical bodies
    _w1, _w2, _w3 : BOOL;
END_VAR

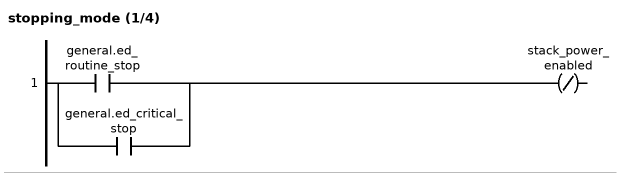
// NETWORK 1
stack_power_enabled := NOT (general.ed_routine_stop OR general.ed_critical_stop);

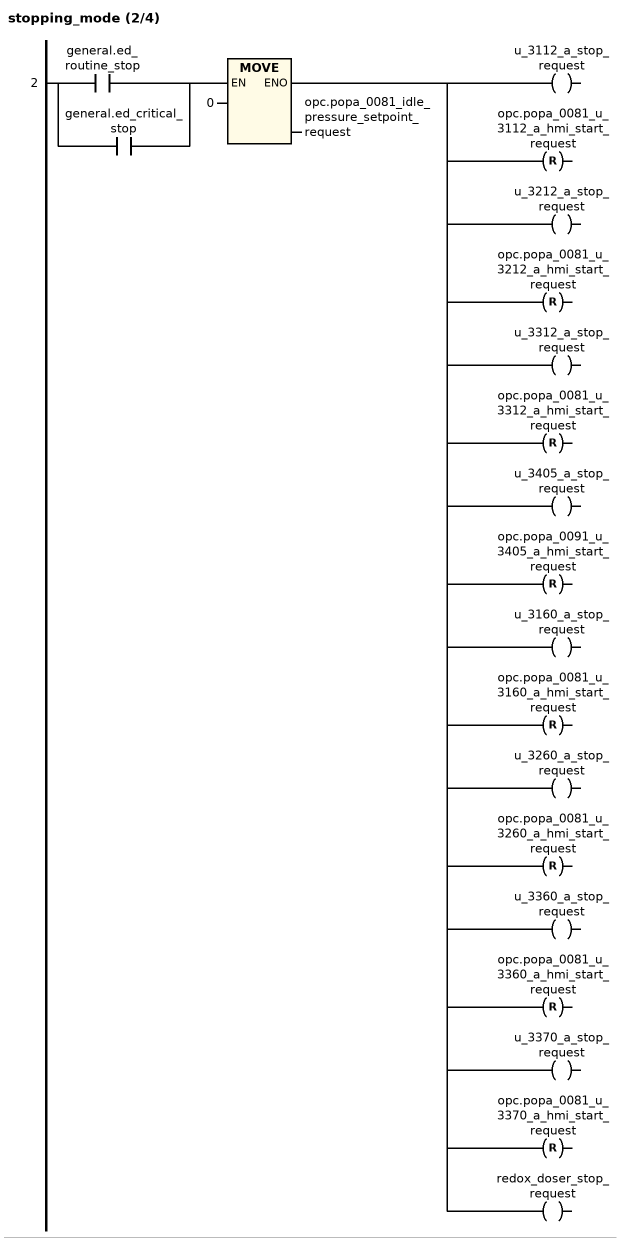
// NETWORK 2
_w1 := general.ed_routine_stop OR general.ed_critical_stop;
IF _w1 THEN opc.popa_0081_idle_pressure_setpoint_request := 0; END_IF
u_3112_a_stop_request := _w1;
opc.popa_0081_u_3112_a_hmi_start_request R= _w1;
u_3212_a_stop_request := _w1;
opc.popa_0081_u_3212_a_hmi_start_request R= _w1;
u_3312_a_stop_request := _w1;
opc.popa_0081_u_3312_a_hmi_start_request R= _w1;
u_3405_a_stop_request := _w1;
opc.popa_0091_u_3405_a_hmi_start_request R= _w1;
u_3160_a_stop_request := _w1;
opc.popa_0081_u_3160_a_hmi_start_request R= _w1;
u_3260_a_stop_request := _w1;
opc.popa_0081_u_3260_a_hmi_start_request R= _w1;
u_3360_a_stop_request := _w1;
opc.popa_0081_u_3360_a_hmi_start_request R= _w1;
u_3370_a_stop_request := _w1;
opc.popa_0081_u_3370_a_hmi_start_request R= _w1;
redox_doser_stop_request := _w1;

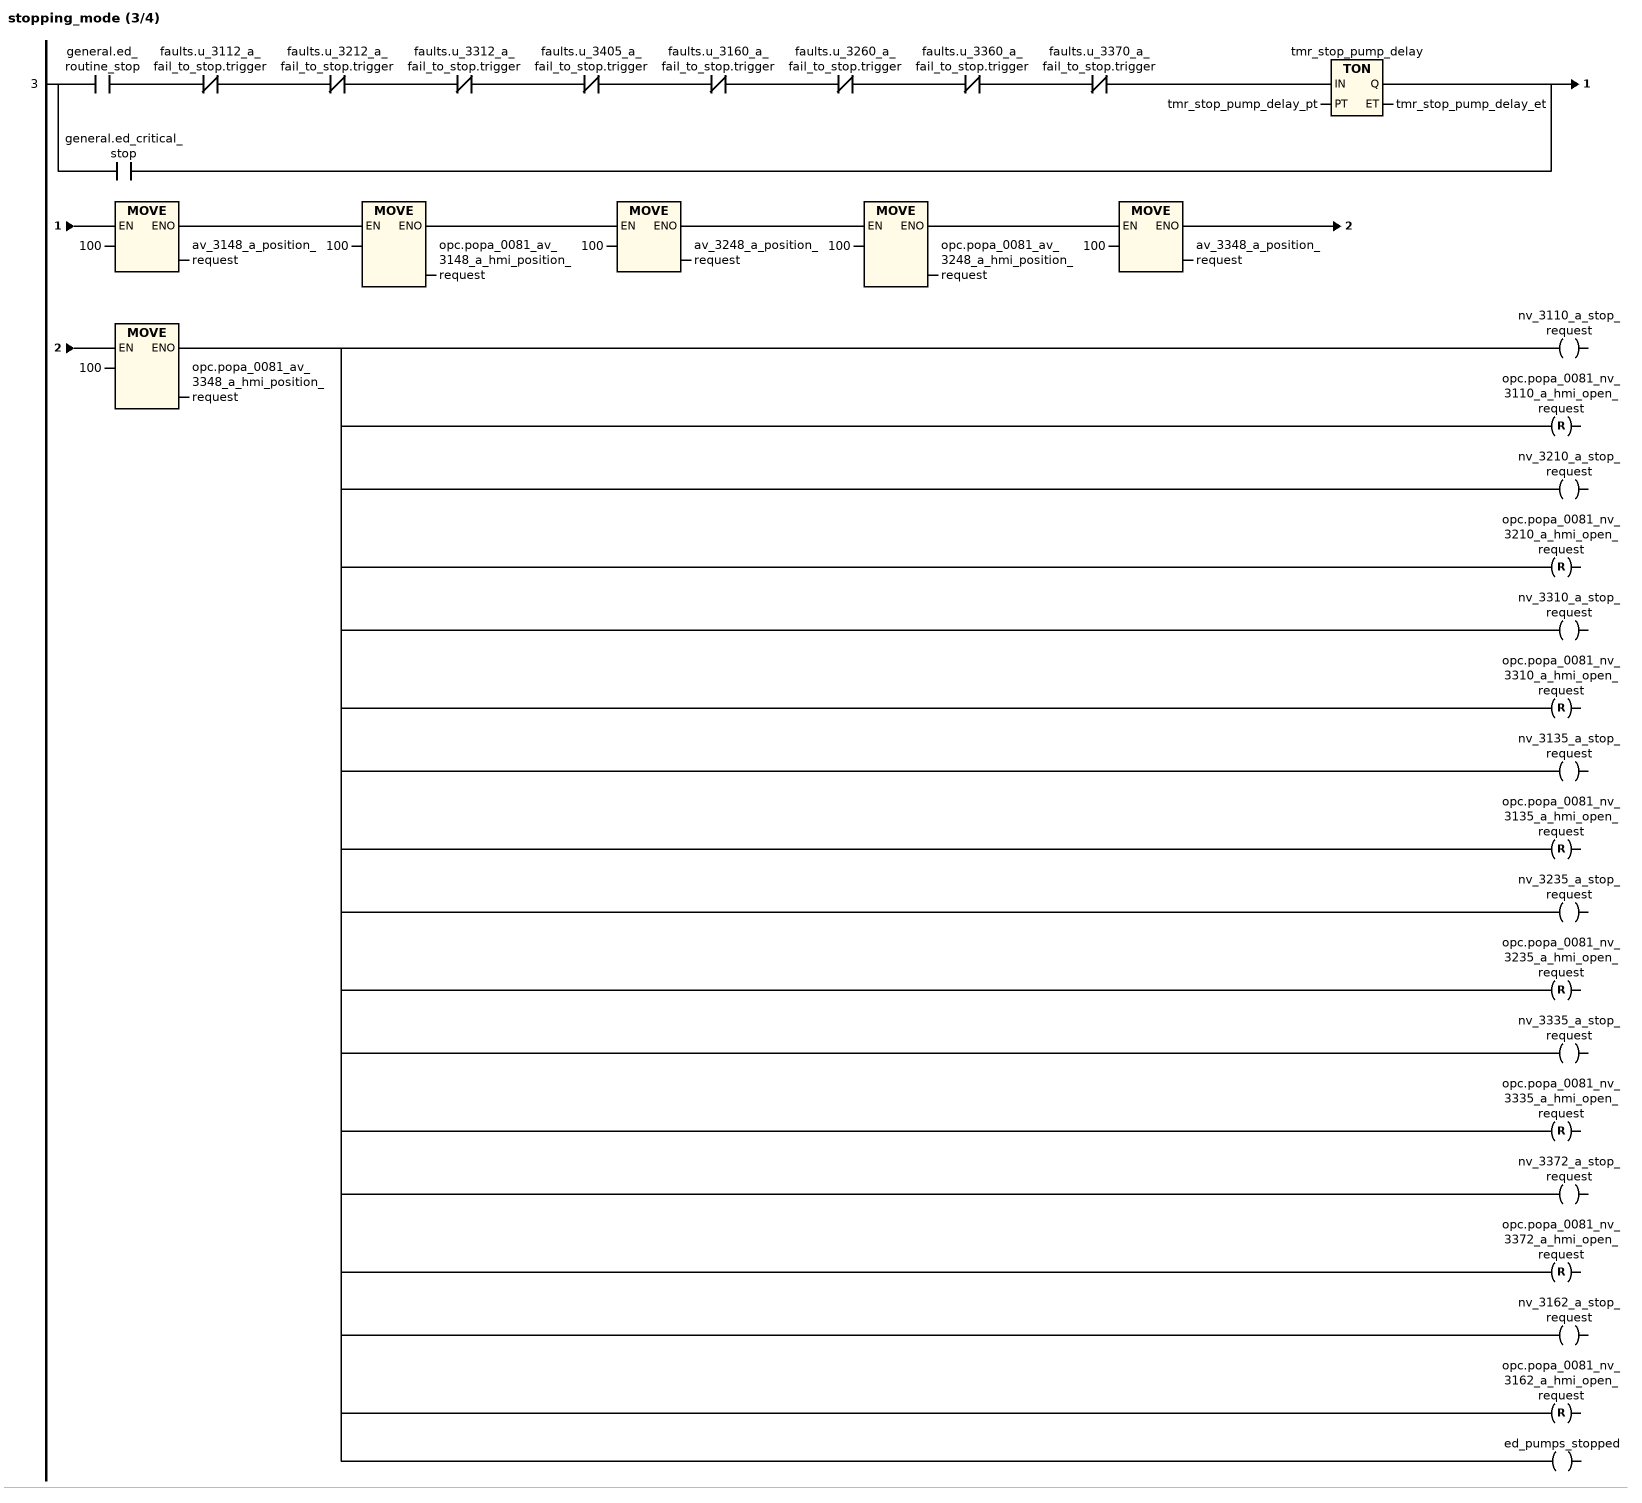
// NETWORK 3
tmr_stop_pump_delay(
    IN := general.ed_routine_stop AND NOT faults.u_3112_a_fail_to_stop.trigger AND NOT faults.u_3212_a_fail_to_stop.trigger AND NOT faults.u_3312_a_fail_to_stop.trigger AND NOT faults.u_3405_a_fail_to_stop.trigger AND NOT faults.u_3160_a_fail_to_stop.trigger AND NOT faults.u_3260_a_fail_to_stop.trigger AND NOT faults.u_3360_a_fail_to_stop.trigger AND NOT faults.u_3370_a_fail_to_stop.trigger,
    PT := tmr_stop_pump_delay_pt,
    ET => tmr_stop_pump_delay_et); // TON
_w2 := tmr_stop_pump_delay.Q OR general.ed_critical_stop;
IF _w2 THEN av_3148_a_position_request := 100; END_IF
IF _w2 THEN opc.popa_0081_av_3148_a_hmi_position_request := 100; END_IF
IF _w2 THEN av_3248_a_position_request := 100; END_IF
IF _w2 THEN opc.popa_0081_av_3248_a_hmi_position_request := 100; END_IF
IF _w2 THEN av_3348_a_position_request := 100; END_IF
IF _w2 THEN opc.popa_0081_av_3348_a_hmi_position_request := 100; END_IF
nv_3110_a_stop_request := _w2;
opc.popa_0081_nv_3110_a_hmi_open_request R= _w2;
nv_3210_a_stop_request := _w2;
opc.popa_0081_nv_3210_a_hmi_open_request R= _w2;
nv_3310_a_stop_request := _w2;
opc.popa_0081_nv_3310_a_hmi_open_request R= _w2;
nv_3135_a_stop_request := _w2;
opc.popa_0081_nv_3135_a_hmi_open_request R= _w2;
nv_3235_a_stop_request := _w2;
opc.popa_0081_nv_3235_a_hmi_open_request R= _w2;
nv_3335_a_stop_request := _w2;
opc.popa_0081_nv_3335_a_hmi_open_request R= _w2;
nv_3372_a_stop_request := _w2;
opc.popa_0081_nv_3372_a_hmi_open_request R= _w2;
nv_3162_a_stop_request := _w2;
opc.popa_0081_nv_3162_a_hmi_open_request R= _w2;
ed_pumps_stopped := _w2;

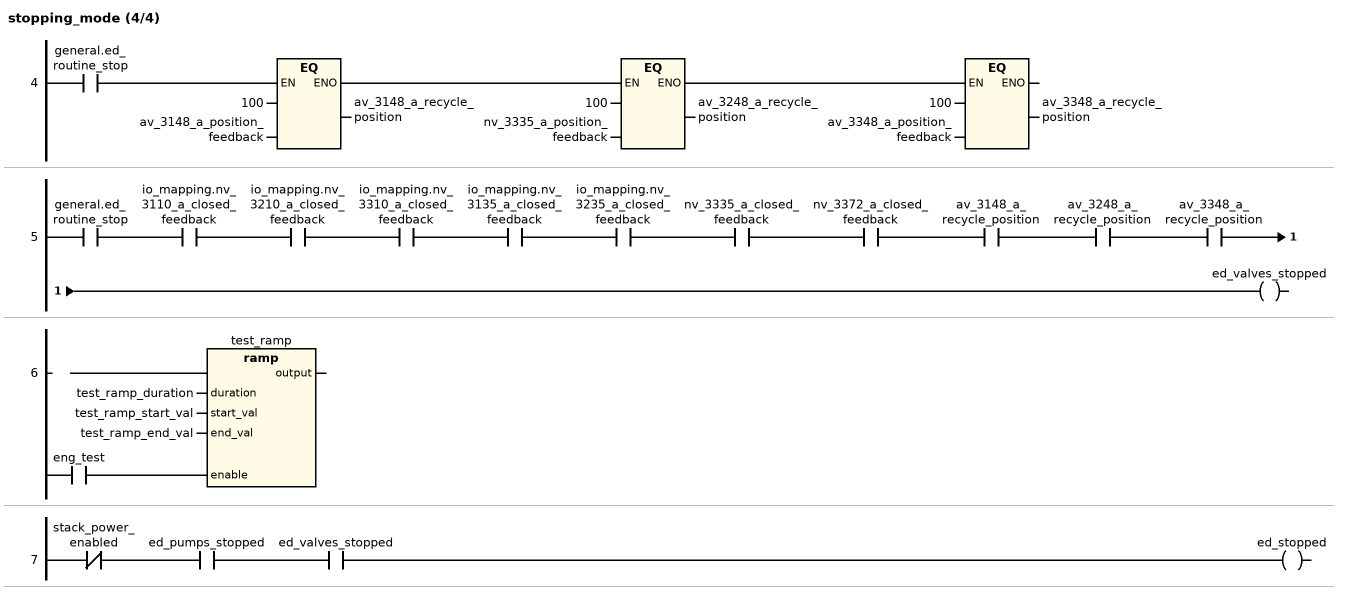
// NETWORK 4
_w3 := general.ed_routine_stop;
IF _w3 THEN av_3148_a_recycle_position := 100 = av_3148_a_position_feedback; END_IF
IF _w3 THEN av_3248_a_recycle_position := 100 = nv_3335_a_position_feedback; END_IF
IF _w3 THEN av_3348_a_recycle_position := 100 = av_3348_a_position_feedback; END_IF

// NETWORK 5
ed_valves_stopped := general.ed_routine_stop AND io_mapping.nv_3110_a_closed_feedback AND io_mapping.nv_3210_a_closed_feedback AND io_mapping.nv_3310_a_closed_feedback AND io_mapping.nv_3135_a_closed_feedback AND io_mapping.nv_3235_a_closed_feedback AND nv_3335_a_closed_feedback AND nv_3372_a_closed_feedback AND av_3148_a_recycle_position AND av_3248_a_recycle_position AND av_3348_a_recycle_position;

// NETWORK 6
test_ramp(
    duration := test_ramp_duration,
    start_val := test_ramp_start_val,
    end_val := test_ramp_end_val,
    enable := eng_test); // ramp

// NETWORK 7
ed_stopped := NOT stack_power_enabled AND ed_pumps_stopped AND ed_valves_stopped;

END_PROGRAM

// ---- POUs/Function Blocks/ramp.TcPOU
FUNCTION_BLOCK PUBLIC ramp
VAR_INPUT
	duration : INT;
	start_val : REAL;
	end_val : REAL;
	enable : BOOL;
END_VAR
VAR_OUTPUT
	output : REAL;
END_VAR
VAR
	ramp_tmr: TON;
	ramp_tmr_et: TIME;
	ramp_counter: CTU;
	ramp_time_delay_ms: real;
	ramp_time_delay: TIME;
	ramp_range : REAL;
	ramp_increment: REAL;
	ramp_tmr_et_ms: REAL;
	ramp_mult_output: REAL;
END_VAR

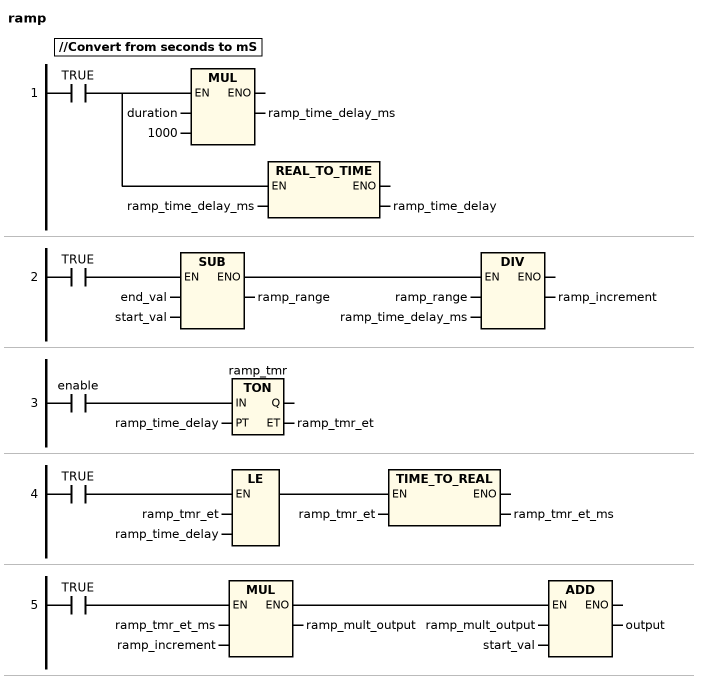
// NETWORK 1
// label: //Convert from seconds to mS
ramp_time_delay_ms := duration * 1000;
ramp_time_delay := REAL_TO_TIME(ramp_time_delay_ms);

// NETWORK 2
ramp_range := end_val - start_val;
ramp_increment := ramp_range / ramp_time_delay_ms;

// NETWORK 3
ramp_tmr(IN := enable, PT := ramp_time_delay, ET => ramp_tmr_et); // TON

// NETWORK 4
IF ramp_tmr_et <= ramp_time_delay THEN ramp_tmr_et_ms := TIME_TO_REAL(ramp_tmr_et); END_IF

// NETWORK 5
ramp_mult_output := ramp_tmr_et_ms * ramp_increment;
output := ramp_mult_output + start_val;

END_FUNCTION_BLOCK

// ---- POUs/cip.TcPOU
PROGRAM cip
VAR
	ed_routine_starting_idle: BOOL;
	idle_redox_doser_enable: BOOL;
	
	tmr_idle_pumps: TON;
	idle_u_3112_a_request: BOOL;
	idle_u_3312_a_request: BOOL;
	idle_u_3405_a_request: BOOL;
	idle_u_3212_a_request: BOOL;
	tmr_idle_pump_delay: TON;
	u_3112_a_running: BOOL;
	u_3112_a_speed_ref: INT;
	u_3112_a_sp: REAL;
	salt_pressure_actual: REAL;
	idle_u_3112_a_ready: BOOL;
	u_3212_a_running: BOOL;
	idle_u_3212_a_ready: BOOL;
	idle_u_3312_a_ready: BOOL;
	u_3312_a_running: BOOL;
	u_3405_a_running: BOOL;
	idle_u_3405_a_ready: BOOL;
	idle_stack_power_enable: BOOL;
	ed_routine_cip: BOOL;
	
		nv_3110_a_open_request: BOOL;
	nv_3210_a_open_request: BOOL;
	nv_3310_a_open_request: BOOL;
	nv_3110_a_open_feedback: BOOL;
	nv_3210_a_open_feedback: BOOL;
	nv_3310_a_open_feedback: BOOL;
	cip_redox_doser_enable: BOOL;
	nv_3372_a_open_request: BOOL;
	nv_3135_a_open_request: BOOL;
	nv_3235_a_open_request: BOOL;
	nv_3335_a_open_request: BOOL;
	nv_3372_a_open_feedback: BOOL;
	nv_3135_a_open_feedback: BOOL;
	nv_3235_a_open_feedback: BOOL;
	nv_3335_a_open_feedback: BOOL;
	tmr_cip_pump_delay: TON;
	idle_u_3370_a_request: BOOL;
	u_3370_a_running: BOOL;
	u_3370_a_sp: REAL;
	tmr_cip_pump_start_delay: TON;
	tmr_cip_run: TON;
	cip_tmr_preset: TIME;
	
	u_3370_a_actual: INT; // What would this be???
	ft_3122_a_tot: INT;
	ft_3222_a_tot: INT;
	ft_3322_a_tot: INT;
	cip_flush_tot: INT;
	cip_flush_sp: INT;
	cip_u_3370_a_request: BOOL;
	cip_complete: BOOL;
	cip_stop_request: BOOL;
	nv_3372_a_cip_request: BOOL;
	nv_3135_a_cip_request: BOOL;
	nv_3235_a_cip_request: BOOL;
	nv_3335_a_cip_request: BOOL;
	redox_doser_cip_enable: BOOL;
	u_3370_a_cip_request: BOOL;
	CIP_TEMP_BIT: BOOL;
	tmr_cip_valve_delay: TON;
	tmr_cip_valve_delay_pt: TIME:= T#30S;
	tmr_cip_valve_delay_et: TIME;
	tmr_cip_valve_delay_q: BOOL;
	u_3112_a_cip_pressure_setpoint_request: REAL;
	u_3370_a_cip_pressure_setpoint_request: REAL;
END_VAR
VAR // added by the converter: edge detectors and wires of the graphical bodies
    _w1, _w2, _w3 : BOOL;
END_VAR

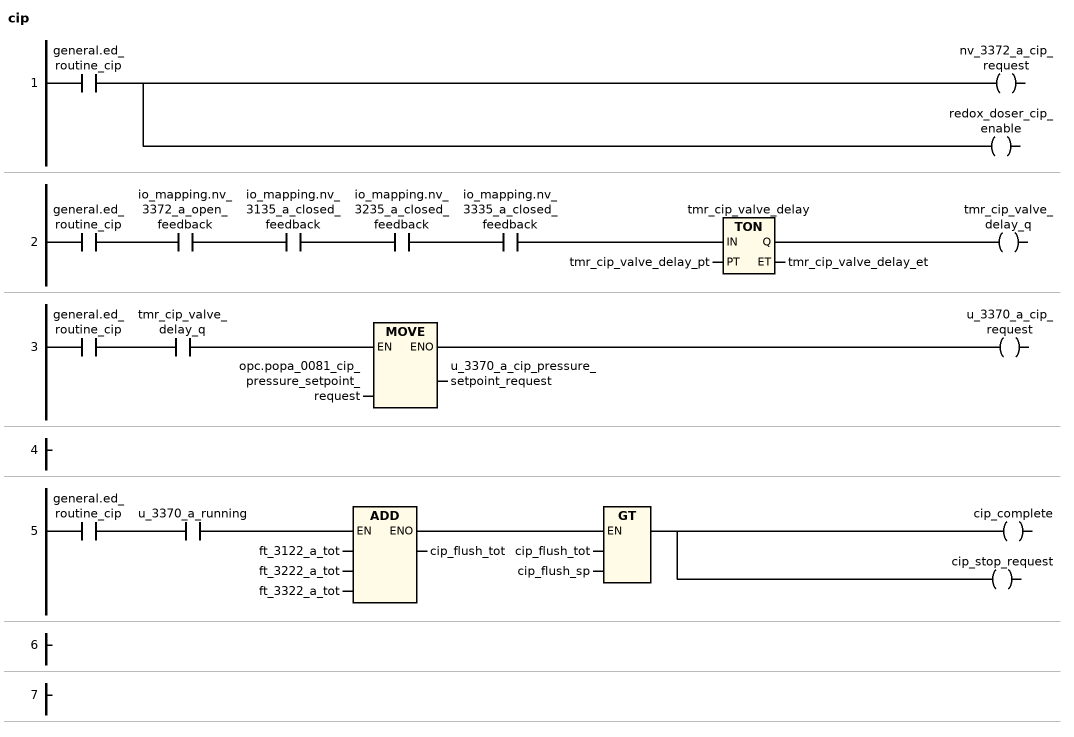
// NETWORK 1
nv_3372_a_cip_request := general.ed_routine_cip;
redox_doser_cip_enable := general.ed_routine_cip;

// NETWORK 2
tmr_cip_valve_delay(
    IN := general.ed_routine_cip AND io_mapping.nv_3372_a_open_feedback AND io_mapping.nv_3135_a_closed_feedback AND io_mapping.nv_3235_a_closed_feedback AND io_mapping.nv_3335_a_closed_feedback,
    PT := tmr_cip_valve_delay_pt,
    ET => tmr_cip_valve_delay_et); // TON
tmr_cip_valve_delay_q := tmr_cip_valve_delay.Q;

// NETWORK 3
_w1 := general.ed_routine_cip AND tmr_cip_valve_delay_q;
IF _w1 THEN u_3370_a_cip_pressure_setpoint_request := opc.popa_0081_cip_pressure_setpoint_request; END_IF
u_3370_a_cip_request := _w1;

// NETWORK 4

// NETWORK 5
_w2 := general.ed_routine_cip AND u_3370_a_running;
IF _w2 THEN cip_flush_tot := ft_3122_a_tot + ft_3222_a_tot + ft_3322_a_tot; END_IF
_w3 := _w2 AND cip_flush_tot > cip_flush_sp;
cip_complete := _w3;
cip_stop_request := _w3;

// NETWORK 6

// NETWORK 7

END_PROGRAM

// ---- POUs/valve_manager.TcPOU
PROGRAM valve_manager
VAR
	//Digital valve
	nv_3110: valve_digital;
	nv_3210: valve_digital;
	nv_3310: valve_digital;
	nv_3135: valve_digital;
	nv_3235: valve_digital;
	nv_3335: valve_digital;
	nv_3372: valve_digital;
	nv_3162: valve_digital;
	
	// Analog Valve Function Block
	av_3148: valve_analog;
	av_3248: valve_analog;
	av_3348: valve_analog;


	//Repeat for each valve?
	u_3112_open_request: BOOL;
	u_3112_idle_request: BOOL;
	u_3112_cip_request: BOOL;
	u_3112_manual_request: BOOL;
	u_3112_stop_request: BOOL;
	u_3112_intlk: BOOL;
	gen_alm_active: BOOL;
	ed_routine_idle: BOOL;
	ed_routine_cip: BOOL;
	ed_routine_manual: BOOL;
	ed_routine_maint: BOOL;
	nv_3110_idle_request: BOOL;
	nv_3110_cip_request: BOOL;
	nv_3110_manual_request: BOOL;
	nv_3110_intlk: BOOL;
	nv_3110_stop_request: BOOL;
	nv_3110_open_request: BOOL;
	nv_3210_open_request: BOOL;
	nv_3310_open_request: BOOL;
	nv_3135_open_request: BOOL;
	nv_3235_open_request: BOOL;
	nv_3335_open_request: BOOL;
	nv_3372_open_request: BOOL;
	nv_3210_idle_request: BOOL;
	nv_3210_cip_request: BOOL;
	nv_3210_manual_request: BOOL;
	nv_3210_stop_request: BOOL;
	nv_3210_intlk: BOOL;
	
	nv_3310_idle_request: BOOL;
	nv_3310_cip_request: BOOL;
	nv_3310_manual_request: BOOL;
	nv_3310_stop_request: BOOL;
	nv_3310_intlk: BOOL;
	
	nv_3135_idle_request: BOOL;
	nv_3135_cip_request: BOOL;
	nv_3135_manual_request: BOOL;
	nv_3135_stop_request: BOOL;
	nv_3135_intlk: BOOL;
	
	nv_3235_idle_request: BOOL;
	nv_3235_cip_request: BOOL;
	nv_3235_manual_request: BOOL;
	nv_3235_stop_request: BOOL;
	nv_3235_intlk: BOOL;
	
	nv_3335_idle_request: BOOL;
	nv_3335_cip_request: BOOL;
	nv_3335_manual_request: BOOL;
	nv_3335_stop_request: BOOL;
	nv_3335_intlk: BOOL;
	
	nv_3372_idle_request: BOOL;
	nv_3372_cip_request: BOOL;
	nv_3372_manual_request: BOOL;
	nv_3372_stop_request: BOOL;
	nv_3372_intlk: BOOL;
	
	nv_3162_idle_request: BOOL;
	nv_3162_cip_request: BOOL;
	nv_3162_manual_request: BOOL;
	nv_3162_stop_request: BOOL;
	nv_3162_intlk: BOOL;
	nv_3162_open_request: BOOL;
	
	av_3148_idle_request: BOOL;
	av_3148_cip_request: BOOL;
	av_3148_idle_position_request: REAL;
	av_3148_position_request: REAL;
	av_3148_cip_position_request: REAL;
	av_3148_manual_position_request: REAL;
	av_3148_manual_request: BOOL;
	av_3148_maint_request: BOOL;
	av_3148_maint_position_request: REAL;
	av_3148_intlk: BOOL;
	av_3148_stop_request: BOOL;
	av_3148_open_request: BOOL;
	
	av_3248_idle_request: BOOL;
	av_3248_cip_request: BOOL;
	av_3248_idle_position_request: REAL;
	av_3248_position_request: REAL;
	av_3248_cip_position_request: REAL;
	av_3248_manual_position_request: REAL;
	av_3248_manual_request: BOOL;
	av_3248_maint_request: BOOL;
	av_3248_maint_position_request: REAL;
	av_3248_intlk: BOOL;
	av_3248_stop_request: BOOL;
	av_3248_open_request: BOOL;
	
	av_3348_idle_request: BOOL;
	av_3348_cip_request: BOOL;
	av_3348_idle_position_request: REAL;
	av_3348_position_request: REAL;
	av_3348_cip_position_request: REAL;
	av_3348_manual_position_request: REAL;
	av_3348_manual_request: BOOL;
	av_3348_maint_request: BOOL;
	av_3348_maint_position_request: REAL;
	av_3348_intlk: BOOL;
	av_3348_stop_request: BOOL;
	av_3348_open_request: BOOL;
	
END_VAR
VAR // added by the converter: edge detectors and wires of the graphical bodies
    _w1, _w2, _w3, _w4, _w5, _w6, _w7, _w8, _w9, _w10, _w11, _w12, _w13, _w14, _w15 : BOOL;
END_VAR

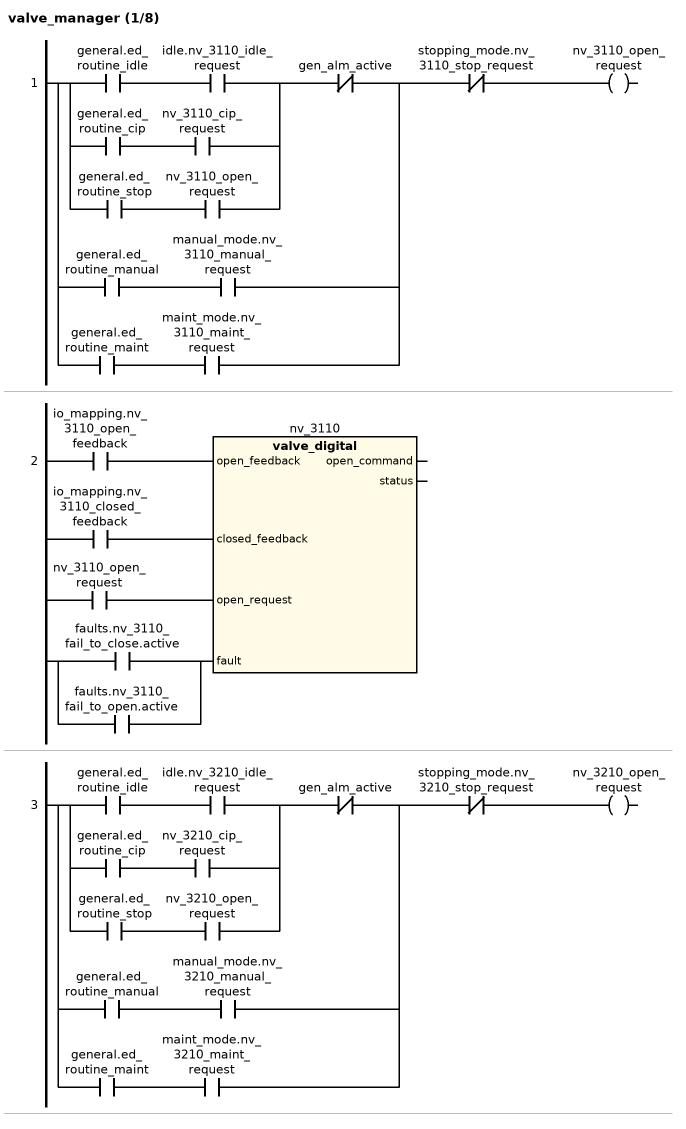
// NETWORK 1
nv_3110_open_request := ((general.ed_routine_idle AND idle.nv_3110_idle_request OR general.ed_routine_cip AND nv_3110_cip_request OR general.ed_routine_stop AND nv_3110_open_request) AND NOT gen_alm_active OR general.ed_routine_manual AND manual_mode.nv_3110_manual_request OR general.ed_routine_maint AND maint_mode.nv_3110_maint_request) AND NOT stopping_mode.nv_3110_stop_request;

// NETWORK 2
nv_3110(
    open_feedback := io_mapping.nv_3110_open_feedback,
    closed_feedback := io_mapping.nv_3110_closed_feedback,
    open_request := nv_3110_open_request,
    fault := faults.nv_3110_fail_to_close.active OR faults.nv_3110_fail_to_open.active); // valve_digital

// NETWORK 3
nv_3210_open_request := ((general.ed_routine_idle AND idle.nv_3210_idle_request OR general.ed_routine_cip AND nv_3210_cip_request OR general.ed_routine_stop AND nv_3210_open_request) AND NOT gen_alm_active OR general.ed_routine_manual AND manual_mode.nv_3210_manual_request OR general.ed_routine_maint AND maint_mode.nv_3210_maint_request) AND NOT stopping_mode.nv_3210_stop_request;

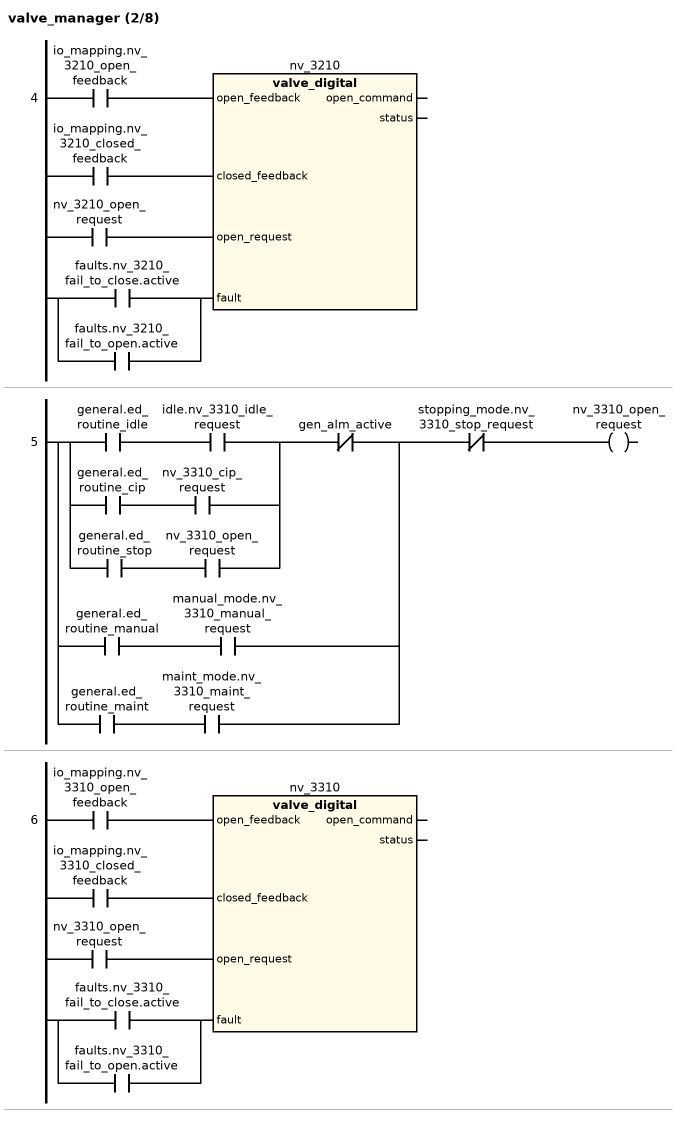
// NETWORK 4
nv_3210(
    open_feedback := io_mapping.nv_3210_open_feedback,
    closed_feedback := io_mapping.nv_3210_closed_feedback,
    open_request := nv_3210_open_request,
    fault := faults.nv_3210_fail_to_close.active OR faults.nv_3210_fail_to_open.active); // valve_digital

// NETWORK 5
nv_3310_open_request := ((general.ed_routine_idle AND idle.nv_3310_idle_request OR general.ed_routine_cip AND nv_3310_cip_request OR general.ed_routine_stop AND nv_3310_open_request) AND NOT gen_alm_active OR general.ed_routine_manual AND manual_mode.nv_3310_manual_request OR general.ed_routine_maint AND maint_mode.nv_3310_maint_request) AND NOT stopping_mode.nv_3310_stop_request;

// NETWORK 6
nv_3310(
    open_feedback := io_mapping.nv_3310_open_feedback,
    closed_feedback := io_mapping.nv_3310_closed_feedback,
    open_request := nv_3310_open_request,
    fault := faults.nv_3310_fail_to_close.active OR faults.nv_3310_fail_to_open.active); // valve_digital

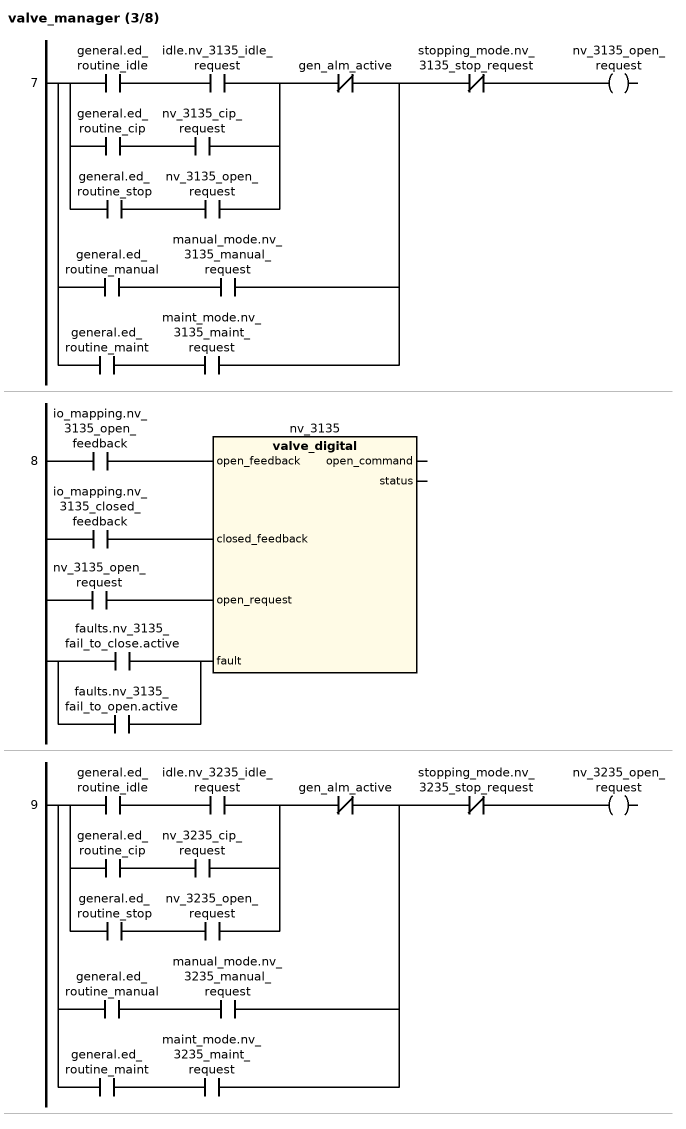
// NETWORK 7
nv_3135_open_request := ((general.ed_routine_idle AND idle.nv_3135_idle_request OR general.ed_routine_cip AND nv_3135_cip_request OR general.ed_routine_stop AND nv_3135_open_request) AND NOT gen_alm_active OR general.ed_routine_manual AND manual_mode.nv_3135_manual_request OR general.ed_routine_maint AND maint_mode.nv_3135_maint_request) AND NOT stopping_mode.nv_3135_stop_request;

// NETWORK 8
nv_3135(
    open_feedback := io_mapping.nv_3135_open_feedback,
    closed_feedback := io_mapping.nv_3135_closed_feedback,
    open_request := nv_3135_open_request,
    fault := faults.nv_3135_fail_to_close.active OR faults.nv_3135_fail_to_open.active); // valve_digital

// NETWORK 9
nv_3235_open_request := ((general.ed_routine_idle AND idle.nv_3235_idle_request OR general.ed_routine_cip AND nv_3235_cip_request OR general.ed_routine_stop AND nv_3235_open_request) AND NOT gen_alm_active OR general.ed_routine_manual AND manual_mode.nv_3235_manual_request OR general.ed_routine_maint AND maint_mode.nv_3235_maint_request) AND NOT stopping_mode.nv_3235_stop_request;

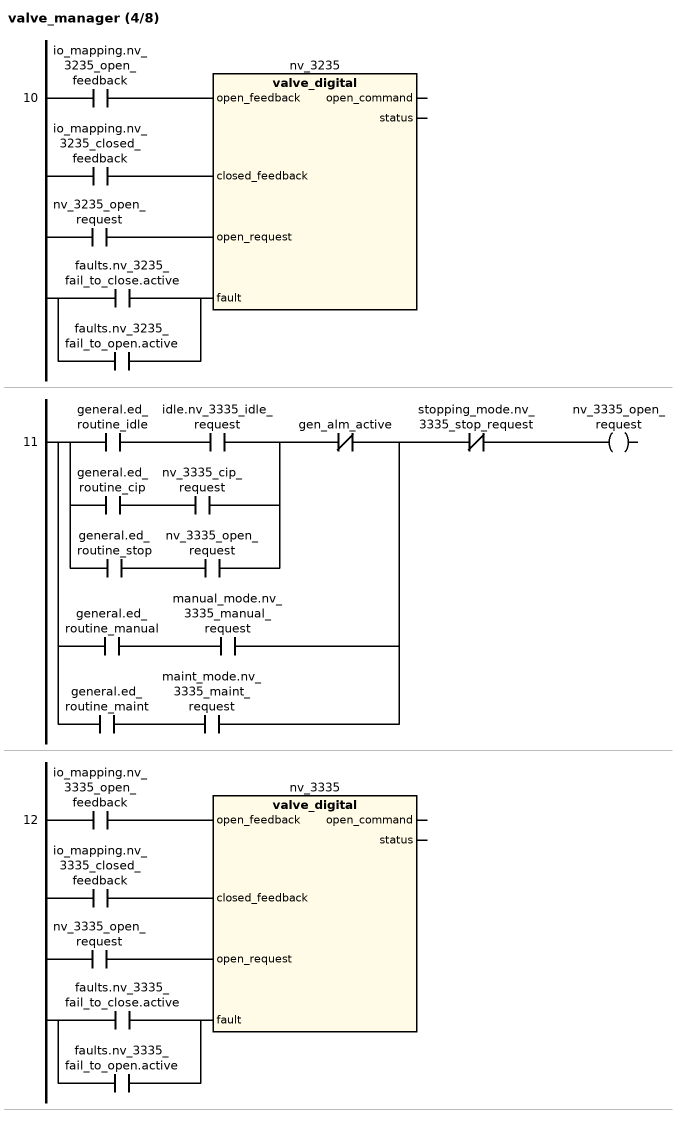
// NETWORK 10
nv_3235(
    open_feedback := io_mapping.nv_3235_open_feedback,
    closed_feedback := io_mapping.nv_3235_closed_feedback,
    open_request := nv_3235_open_request,
    fault := faults.nv_3235_fail_to_close.active OR faults.nv_3235_fail_to_open.active); // valve_digital

// NETWORK 11
nv_3335_open_request := ((general.ed_routine_idle AND idle.nv_3335_idle_request OR general.ed_routine_cip AND nv_3335_cip_request OR general.ed_routine_stop AND nv_3335_open_request) AND NOT gen_alm_active OR general.ed_routine_manual AND manual_mode.nv_3335_manual_request OR general.ed_routine_maint AND maint_mode.nv_3335_maint_request) AND NOT stopping_mode.nv_3335_stop_request;

// NETWORK 12
nv_3335(
    open_feedback := io_mapping.nv_3335_open_feedback,
    closed_feedback := io_mapping.nv_3335_closed_feedback,
    open_request := nv_3335_open_request,
    fault := faults.nv_3335_fail_to_close.active OR faults.nv_3335_fail_to_open.active); // valve_digital

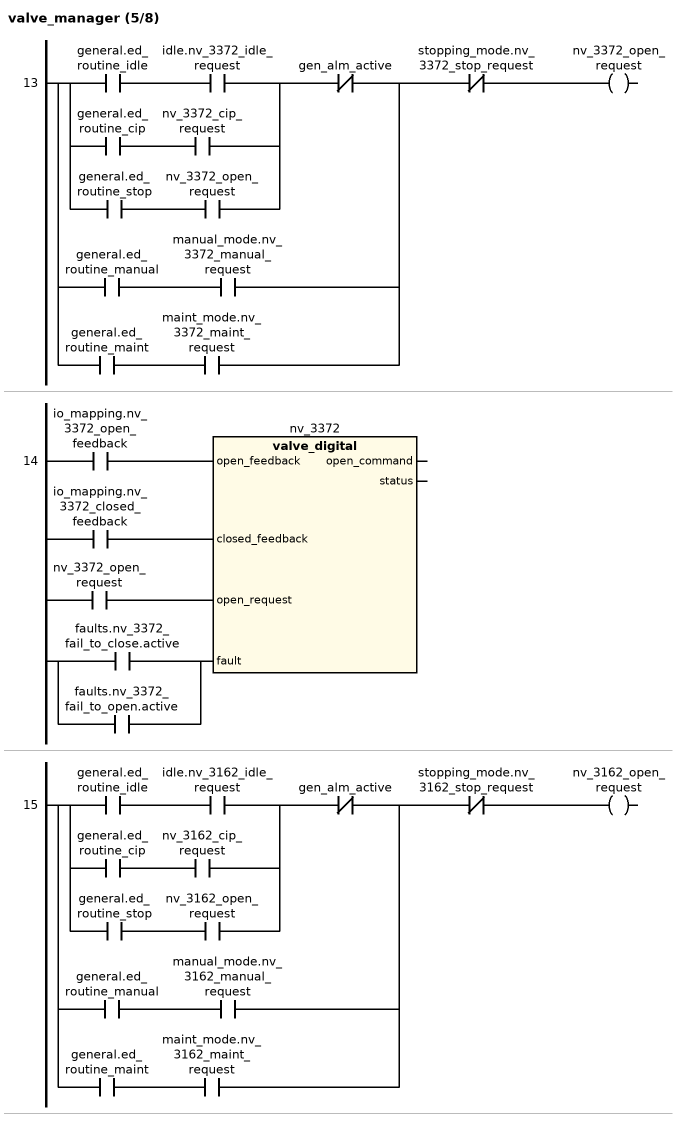
// NETWORK 13
nv_3372_open_request := ((general.ed_routine_idle AND idle.nv_3372_idle_request OR general.ed_routine_cip AND nv_3372_cip_request OR general.ed_routine_stop AND nv_3372_open_request) AND NOT gen_alm_active OR general.ed_routine_manual AND manual_mode.nv_3372_manual_request OR general.ed_routine_maint AND maint_mode.nv_3372_maint_request) AND NOT stopping_mode.nv_3372_stop_request;

// NETWORK 14
nv_3372(
    open_feedback := io_mapping.nv_3372_open_feedback,
    closed_feedback := io_mapping.nv_3372_closed_feedback,
    open_request := nv_3372_open_request,
    fault := faults.nv_3372_fail_to_close.active OR faults.nv_3372_fail_to_open.active); // valve_digital

// NETWORK 15
nv_3162_open_request := ((general.ed_routine_idle AND idle.nv_3162_idle_request OR general.ed_routine_cip AND nv_3162_cip_request OR general.ed_routine_stop AND nv_3162_open_request) AND NOT gen_alm_active OR general.ed_routine_manual AND manual_mode.nv_3162_manual_request OR general.ed_routine_maint AND maint_mode.nv_3162_maint_request) AND NOT stopping_mode.nv_3162_stop_request;

